// TIA Portal project "Szklarnia_AMN_V15.1" (V15.1)

(* hardware
DEVICE "S7-1200 station_1"  S7-1200 Station
   slot 0: "Rack_0"  Rack  V1.0
   slot 1: "PLC_1"  CPU 1212C AC/DC/Rly  6ES7 212-1BD30-0XB0  V2.2
   slot 101: "CM 1241 (RS232)_1"  6ES7 241-1AH30-0XB0  V1.0
DEVICE "HMI_1"  KTP600 Basic color PN
   slot 0: "HMI"  HMI  6AV6 647-0AD11-3AX0  12.0.0.0
   slot 1: "HMI_RT_1"  KTP600 Basic color PN  6AV6 647-0AD11-3AX0  12.0.0.0
   slot 5: "HMI_1.IE_CP_1"  PROFINET Interface
      slot 1: "PROFINET Interface_1"  PROFINET Interface
         slot 1: "Port_1"  Port
*)

// ===== PLC "PLC_1"  CPU 1212C AC/DC/Rly =====

VAR_GLOBAL   // PLC tag table "Default tag table"
   "System_Byte" AT %MB1 : Byte;
   "FirstScan" AT %M1.0 : Bool;
   "DiagStatusUpdate" AT %M1.1 : Bool;
   "AlwaysTRUE" AT %M1.2 : Bool;
   "AlwaysFALSE" AT %M1.3 : Bool;
   "Clock_Byte" AT %MB0 : Byte;
   "Clock_10Hz" AT %M0.0 : Bool;
   "Clock_5Hz" AT %M0.1 : Bool;
   "Clock_2.5Hz" AT %M0.2 : Bool;
   "Clock_2Hz" AT %M0.3 : Bool;
   "Clock_1.25Hz" AT %M0.4 : Bool;
   "Clock_1Hz" AT %M0.5 : Bool;
   "Clock_0.625Hz" AT %M0.6 : Bool;
   "Clock_0.5Hz" AT %M0.7 : Bool;
   "Sensor_nasłonecznienia" AT %IW64 : Word;
   "Tag_2" AT %I0.0 : Bool;
   "Rolety" AT %Q0.0 : Bool;
   "Czujnik" AT %IW66 : Int;
   "Okna" AT %Q0.1 : Bool;
   "Pompa_zbiornik" AT %Q0.2 : Bool;
   "Pompa_sieć" AT %Q0.3 : Bool;
   "Nawadnianie_strefa_1" AT %Q0.4 : Bool;
   "Nawadnianie_strefa_2" AT %Q0.5 : Bool;
   "Nawadnianie_strefa_3" AT %Q0.6 : Bool;
   "Nawadnianie_strefa_4" AT %Q0.7 : Bool;
END_VAR

DATA_BLOCK "Naslonecznienie_DB"   // DB1
{ S7_Optimized_Access := 'TRUE' }
AUTHOR : AMN
VERSION : 0.1
// stored: InstanceOfName Naslonecznienie
"Naslonecznienie"
BEGIN
END_DATA_BLOCK

DATA_BLOCK "Dane_programu"   // DB2
TITLE = Dane - zmienne
{ S7_Optimized_Access := 'TRUE' }
AUTHOR : AMN
VERSION : 0.1
// Zmienne dostępne dla całego programu.
   VAR
      blindShut : Bool := false;   // Stan rolet: 1 - zasłonięte, 0 - odsłonięte.
      Light_Lux_temp : Real;   // Wartość pomocnicza do działania programu - nasłonecznienie.
      lightLux_ : Real := 0.0;   // Nasłonecznienie.
      Temp_ : Real := 0.0;   // Temperatura.
      CO2_ : Real := 0.0;   // Poziom CO2.
      setCO2 : Real := 5.0;   // Docelowa wartość CO2.
      setCO2_ : Real := 50.0;   // Docelowa wartość CO2 z HMI.
      setTemp : Real := 5.0;   // Docelowa wartość temperatury.
      setTemp_ : Real := 50.0;   // Docelowa wartość temperatury z HMI.
      StopBtn : Bool := false;   // Wyłącznik awaryjny: 1 - aktywny (blokada wszytskiego), 0 - nieaktywny.
      WaterLevel : Real := 5.0;   // Minimalny poziom wody w zbiorniku.
      StopPodlewanie : Bool := false;   // Blokada podlewania stref: 1 - Blokada podlewania, 0 - Możliwe podlewanie.
      Strefa1 : Bool := false;   // Blokada podlewania strefy 1: 1 - Blokada podlewania, 0 - możliwe podlewanie.
      Strefa2 : Bool := false;   // Blokada podlewania strefy 2: 1 - Blokada podlewania, 0 - możliwe podlewanie.
      Strefa3 : Bool := false;   // Blokada podlewania strefy 3: 1 - Blokada podlewania, 0 - możliwe podlewanie.
      Strefa4 : Bool := false;   // Blokada podlewania strefy 4: 1 - Blokada podlewania, 0 - możliwe podlewanie.
      Strefa5 : Bool := false;   // Blokada podlewania strefy 5: 1 - Blokada podlewania, 0 - możliwe podlewanie.
      setHum_Strefa2 : Real := 5.0;   // Docelowa wartość wilgotności - Strefa 2.
      setHum_Strefa1 : Real := 5.0;   // Docelowa wartość wilgotności - Strefa 1.
      setHum_Strefa5 : Real := 5.0;   // Docelowa wartość wilgotności - Strefa 5.
      setHum_Strefa4 : Real := 5.0;   // Docelowa wartość wilgotności - Strefa 4.
      setHum_Strefa3 : Real := 5.0;   // Docelowa wartość wilgotności - Strefa 3.
      setHum_Strefa1_ : Real := 50.0;   // Docelowa wartość wilgotności z HMI - Strefa 1.
      setHum_Strefa2_ : Real := 50.0;   // Docelowa wartość wilgotności z HMI - Strefa 2.
      setHum_Strefa3_ : Real := 50.0;   // Docelowa wartość wilgotności z HMI - Strefa 3.
      setHum_Strefa4_ : Real := 50.0;   // Docelowa wartość wilgotności z HMI - Strefa 4.
      setHum_Strefa5_ : Real := 50.0;   // Docelowa wartość wilgotności z HMI - Strefa 5.
      Strefa1_podlewanie : Bool := false;   // Aktywne podlewanie strefy 1: 1 - podlewanie, 0 - nie podlewa.
      Strefa2_podlewanie : Bool := false;   // Aktywne podlewanie strefy 2: 1 - podlewanie, 0 - nie podlewa.
      Strefa3_podlewanie : Bool := false;   // Aktywne podlewanie strefy 3: 1 - podlewanie, 0 - nie podlewa.
      Strefa4_podlewanie : Bool := false;   // Aktywne podlewanie strefy 4: 1 - podlewanie, 0 - nie podlewa.
      Strefa5_podlewanie : Bool := false;   // Aktywne podlewanie strefy 5: 1 - podlewanie, 0 - nie podlewa.
      WinOpen : Bool := false;   // Stan okien: 1 - otwarte, 0 - zamknięte.
      setLux : Real := 5.0;   // Docelowa wartość oświetlenia.
      setLux_ : Real := 50.0;   // Docelowa wartość oświetlenia z HMI.
      Hum_Strefa5 : Real := 0.0;   // Wilgotność strefy 5.
      Hum_Strefa4 : Real := 0.0;   // Wilgotność strefy 4.
      Hum_Strefa3 : Real := 0.0;   // Wilgotność strefy 3.
      Hum_Strefa2 : Real := 0.0;   // Wilgotność strefy 2.
      Hum_Strefa1 : Real := 0.0;   // Wilgotność strefy 1.
      Lux_Start : Bool := true;   // Pomiar początkowy nasłonecznienia.
      Nasłonecznienie : Array[0..6] of Real;   // Akwizycja pomiarów do wizualizacji - nałonecznienie.
      CO2 : Array[0..6] of Real;   // Akwizycja pomiarów do wizualizacji - CO2.
      Temperatura : Array[0..6] of Real;   // Akwizycja pomiarów do wizualizacji - Temperatura.
      Hum_1 : Array[0..6] of Real;   // Akwizycja pomiarów do wizualizacji - wilgotność strefy 1.
      Hum_2 : Array[0..6] of Real;   // Akwizycja pomiarów do wizualizacji - wilgotność strefy 2.
      Hum_3 : Array[0..6] of Real;   // Akwizycja pomiarów do wizualizacji - wilgotność strefy 3.
      Hum_4 : Array[0..6] of Real;   // Akwizycja pomiarów do wizualizacji - wilgotność strefy 4.
      Hum_5 : Array[0..6] of Real;   // Akwizycja pomiarów do wizualizacji - wilgotność strefy 5.
   END_VAR
BEGIN
   Nasłonecznienie[0] := 30.0;
   Nasłonecznienie[1] := 35.0;
   Nasłonecznienie[2] := 70.0;
   Nasłonecznienie[3] := 60.0;
   Nasłonecznienie[4] := 75.0;
   Nasłonecznienie[5] := 25.0;
   Nasłonecznienie[6] := 10.0;
   CO2[0] := 10.0;
   CO2[1] := 11.0;
   CO2[2] := 15.0;
   CO2[3] := 8.0;
   CO2[4] := 7.0;
   CO2[5] := 10.0;
   CO2[6] := 11.0;
   Temperatura[0] := 15.0;
   Temperatura[1] := 16.0;
   Temperatura[2] := 20.0;
   Temperatura[3] := 19.0;
   Temperatura[4] := 21.0;
   Temperatura[5] := 22.2;
   Temperatura[6] := 23.4;
   Hum_1[0] := 10.0;
   Hum_1[1] := 20.0;
   Hum_1[2] := 30.0;
   Hum_1[3] := 40.0;
   Hum_1[4] := 50.0;
   Hum_1[5] := 50.0;
   Hum_1[6] := 60.0;
   Hum_2[0] := 90.0;
   Hum_2[1] := 80.0;
   Hum_2[2] := 44.4;
   Hum_2[3] := 34.3;
   Hum_2[4] := 77.7;
   Hum_2[5] := 78.8;
   Hum_2[6] := 80.0;
   Hum_3[0] := 33.3;
   Hum_3[1] := 56.6;
   Hum_3[2] := 76.7;
   Hum_3[3] := 87.8;
   Hum_3[4] := 98.9;
   Hum_3[5] := 12.1;
   Hum_3[6] := 45.4;
   Hum_4[0] := 66.6;
   Hum_4[1] := 77.7;
   Hum_4[2] := 65.6;
   Hum_4[3] := 55.5;
   Hum_4[4] := 55.5;
   Hum_4[5] := 55.5;
   Hum_4[6] := 66.4;
   Hum_5[0] := 23.4;
   Hum_5[1] := 34.5;
   Hum_5[2] := 53.5;
   Hum_5[3] := 98.7;
   Hum_5[4] := 54.3;
   Hum_5[5] := 56.9;
   Hum_5[6] := 22.2;
END_DATA_BLOCK

DATA_BLOCK "CO2_DB"   // DB8
{ S7_Optimized_Access := 'TRUE' }
AUTHOR : AMN
VERSION : 0.1
// stored: InstanceOfName CO2
"CO2"
BEGIN
END_DATA_BLOCK

DATA_BLOCK "Naslonecznienie_DB_1"   // DB9
{ S7_Optimized_Access := 'TRUE' }
AUTHOR : AMN
VERSION : 0.1
// stored: InstanceOfName Naslonecznienie
"Naslonecznienie"
BEGIN
END_DATA_BLOCK

DATA_BLOCK "CO2_DB_1"   // DB10
{ S7_Optimized_Access := 'TRUE' }
AUTHOR : AMN
VERSION : 0.1
// stored: InstanceOfName CO2
"CO2"
BEGIN
END_DATA_BLOCK

DATA_BLOCK "Temperature_DB"   // DB11
{ S7_Optimized_Access := 'TRUE' }
AUTHOR : AMN
VERSION : 0.1
// stored: InstanceOfName Temperature
"Temperature"
BEGIN
END_DATA_BLOCK

DATA_BLOCK "Nawadniane_DB"   // DB12
{ S7_Optimized_Access := 'TRUE' }
AUTHOR : AMN
VERSION : 0.1
// stored: InstanceOfName Nawadniane
"Nawadniane"
BEGIN
END_DATA_BLOCK

DATA_BLOCK "Nawadniane_DB_1"   // DB13
{ S7_Optimized_Access := 'TRUE' }
AUTHOR : AMN
VERSION : 0.1
// stored: InstanceOfName Nawadniane
"Nawadniane"
BEGIN
END_DATA_BLOCK

DATA_BLOCK "Nawadniane_DB_2"   // DB14
{ S7_Optimized_Access := 'TRUE' }
AUTHOR : AMN
VERSION : 0.1
// stored: InstanceOfName Nawadniane
"Nawadniane"
BEGIN
END_DATA_BLOCK

DATA_BLOCK "Nawadniane_DB_3"   // DB15
{ S7_Optimized_Access := 'TRUE' }
AUTHOR : AMN
VERSION : 0.1
// stored: InstanceOfName Nawadniane
"Nawadniane"
BEGIN
END_DATA_BLOCK

DATA_BLOCK "Nawadniane_DB_4"   // DB16
{ S7_Optimized_Access := 'TRUE' }
AUTHOR : AMN
VERSION : 0.1
// stored: InstanceOfName Nawadniane
"Nawadniane"
BEGIN
END_DATA_BLOCK

// folder: System blocks/Program resources

DATA_BLOCK "IEC_Timer_0_DB"   // DB3
{ S7_Optimized_Access := 'TRUE' }
AUTHOR : Simatic
FAMILY : IEC
NAME : IEC_TMR
VERSION : 1.0
// stored: InstanceOfName IEC_TIMER
"IEC_TIMER"
BEGIN
END_DATA_BLOCK

DATA_BLOCK "IEC_Timer_0_DB_1"   // DB4
{ S7_Optimized_Access := 'TRUE' }
AUTHOR : Simatic
FAMILY : IEC
NAME : IEC_TMR
VERSION : 1.0
// stored: InstanceOfName IEC_TIMER
"IEC_TIMER"
BEGIN
END_DATA_BLOCK

DATA_BLOCK "IEC_Timer_0_DB_2"   // DB5
{ S7_Optimized_Access := 'TRUE' }
AUTHOR : Simatic
FAMILY : IEC
NAME : IEC_TMR
VERSION : 1.0
// stored: InstanceOfName IEC_TIMER
"IEC_TIMER"
BEGIN
END_DATA_BLOCK

DATA_BLOCK "IEC_Timer_0_DB_3"   // DB6
{ S7_Optimized_Access := 'TRUE' }
AUTHOR : Simatic
FAMILY : IEC
NAME : IEC_TMR
VERSION : 1.0
// stored: InstanceOfName IEC_TIMER
"IEC_TIMER"
BEGIN
END_DATA_BLOCK

DATA_BLOCK "IEC_Timer_0_DB_4"   // DB7
{ S7_Optimized_Access := 'TRUE' }
AUTHOR : Simatic
FAMILY : IEC
NAME : IEC_TMR
VERSION : 1.0
// stored: InstanceOfName IEC_TIMER
"IEC_TIMER"
BEGIN
END_DATA_BLOCK

DATA_BLOCK "IEC_Timer_0_DB_5"   // DB17
{ S7_Optimized_Access := 'TRUE' }
AUTHOR : Simatic
FAMILY : IEC
NAME : IEC_TMR
VERSION : 1.0
// stored: InstanceOfName IEC_TIMER
"IEC_TIMER"
BEGIN
END_DATA_BLOCK

// folder: (top level)

FUNCTION_BLOCK "Naslonecznienie"   // FB1, LAD
TITLE = Naslonecznienie - rolety
{ S7_Optimized_Access := 'TRUE' }
AUTHOR : AMN
VERSION : 0.1
// Blok sterowania nasłonecznieniem - rolety
   VAR_INPUT
      lightLux_sensor : Int;
   END_VAR
   VAR_OUTPUT
      Rolety : Bool;   // True - zasłonięte, False - odsłonięte
   END_VAR
   VAR_TEMP
      lightLux_norm : Real;
      Galaz_TAK : Bool;
      lightLux : Real;
   END_VAR
   VAR_TEMP   // added for the SCL form of the ladder/FBD networks
      _w1 : Bool;
      _w2 : Bool;
   END_VAR
BEGIN

REGION Network 1: Odczytanie nasłoncznienia
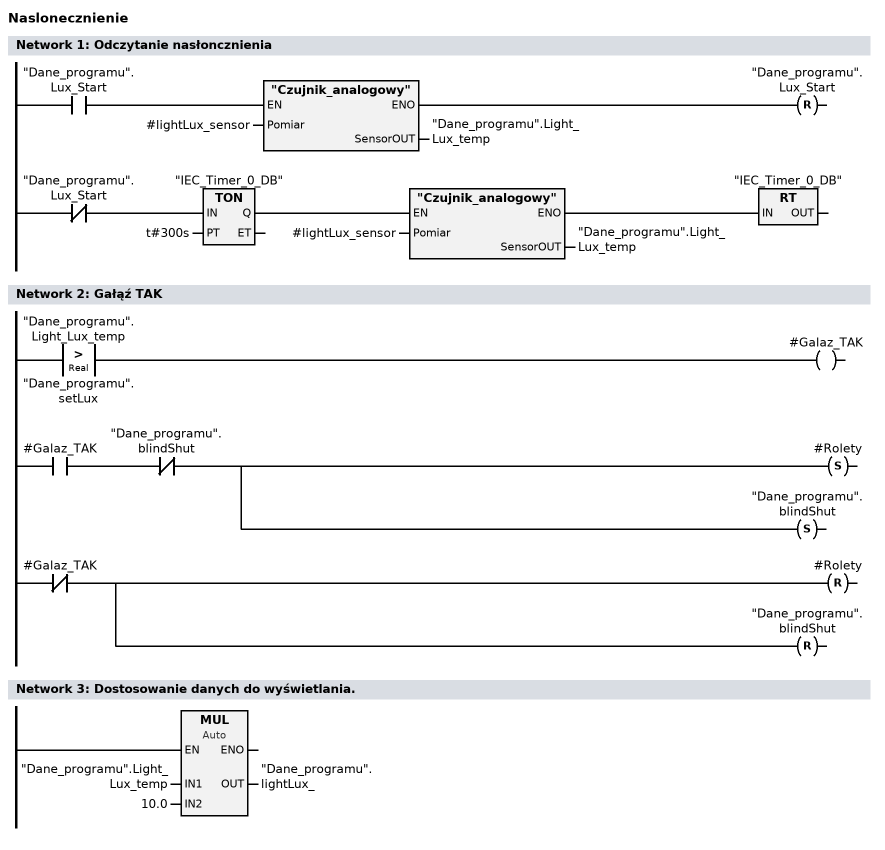
   "Czujnik_analogowy"(EN := "Dane_programu".Lux_Start,
                       Pomiar := #lightLux_sensor,
                       SensorOUT => "Dane_programu".Light_Lux_temp,
                       ENO => #_w1);
   IF #_w1 THEN "Dane_programu".Lux_Start := FALSE; END_IF;
   "IEC_Timer_0_DB".TON(IN := NOT "Dane_programu".Lux_Start, PT := t#300s);
   "Czujnik_analogowy"(EN := "IEC_Timer_0_DB".Q,
                       Pomiar := #lightLux_sensor,
                       SensorOUT => "Dane_programu".Light_Lux_temp,
                       ENO => #_w2);
   IF #_w2 THEN RESET_TIMER("IEC_Timer_0_DB"); END_IF;
END_REGION

REGION Network 2: Gałąź TAK
   RUNG wire#powerrail
      { S7_Templates := "SrcType := Real" } GT_Contact(in1 := "Dane_programu".Light_Lux_temp, in2 := "Dane_programu".setLux)
      Coil( #Galaz_TAK )
   END_RUNG
   RUNG wire#powerrail
      Contact( #Galaz_TAK )
      I_Contact( "Dane_programu".blindShut )
      wire#w1
      S_Coil( #Rolety )
   END_RUNG
   RUNG wire#w1
      S_Coil( "Dane_programu".blindShut )
   END_RUNG
   RUNG wire#powerrail
      I_Contact( #Galaz_TAK )
      wire#w2
      R_Coil( #Rolety )
   END_RUNG
   RUNG wire#w2
      R_Coil( "Dane_programu".blindShut )
   END_RUNG
   // the same network as SCL:
   #Galaz_TAK := "Dane_programu".Light_Lux_temp > "Dane_programu".setLux;
   IF #Galaz_TAK AND NOT "Dane_programu".blindShut THEN
       #Rolety := TRUE;
       "Dane_programu".blindShut := TRUE;
   END_IF;
   IF NOT #Galaz_TAK THEN
       #Rolety := FALSE;
       "Dane_programu".blindShut := FALSE;
   END_IF;
END_REGION

REGION Network 3: Dostosowanie danych do wyświetlania.
   RUNG wire#powerrail
      { S7_GenerateENO := "TRUE" } Mul(in1 := "Dane_programu".Light_Lux_temp, in2 := 10.0, out => "Dane_programu".lightLux_)
   END_RUNG
   // the same network as SCL:
   "Dane_programu".lightLux_ := "Dane_programu".Light_Lux_temp * 10.0;
END_REGION
END_FUNCTION_BLOCK

FUNCTION_BLOCK "CO2"   // FB2, LAD
TITLE = Sterowanie CO2
{ S7_Optimized_Access := 'TRUE' }
AUTHOR : AMN
VERSION : 0.1
// Schemat sterowania poziomem CO2
   VAR_INPUT
      CO2Sensor : Int;
   END_VAR
   VAR_OUTPUT
      Windows : Bool;   // True - otwarte, False - zamknięte
   END_VAR
   VAR_TEMP
      CO2_mes : Real;   // Wartość poziomu CO2
      temp1 : Bool;
      WinFlag : Bool;
   END_VAR
   VAR_TEMP   // added for the SCL form of the ladder/FBD networks
      _w1 : Bool;
   END_VAR
BEGIN

REGION Network 1
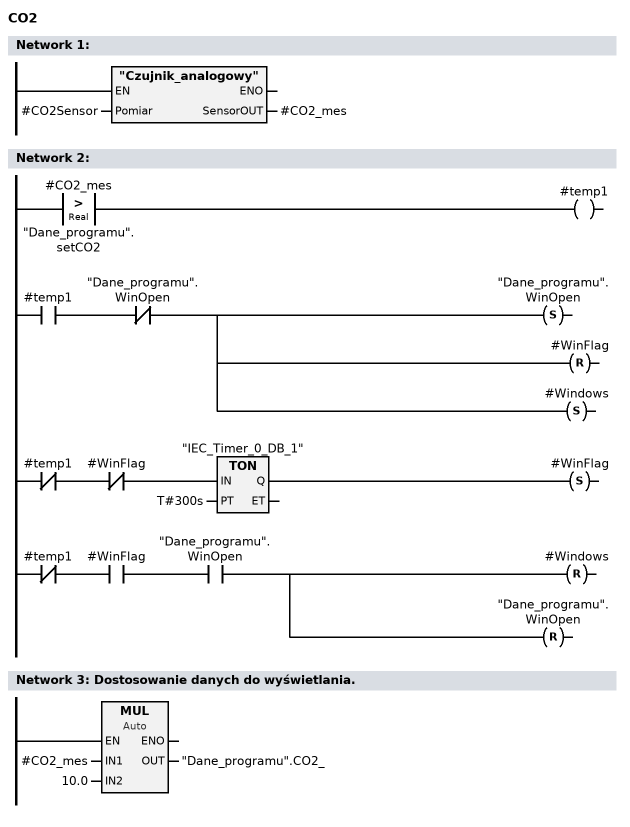
   RUNG wire#powerrail
      "Czujnik_analogowy"(Pomiar := #CO2Sensor, SensorOUT => #CO2_mes)
   END_RUNG
   // the same network as SCL:
   "Czujnik_analogowy"(Pomiar := #CO2Sensor, SensorOUT => #CO2_mes);
END_REGION

REGION Network 2
   #temp1 := #CO2_mes > "Dane_programu".setCO2;
   #_w1 := #temp1 AND NOT "Dane_programu".WinOpen;
   IF #_w1 THEN
       "Dane_programu".WinOpen := TRUE;
       #WinFlag := FALSE;
       #Windows := TRUE;
   END_IF;
   "IEC_Timer_0_DB_1".TON(IN := NOT #temp1 AND NOT #WinFlag, PT := T#300s);
   IF "IEC_Timer_0_DB_1".Q THEN #WinFlag := TRUE; END_IF;
   IF NOT #temp1 AND #WinFlag AND "Dane_programu".WinOpen THEN
       #Windows := FALSE;
       "Dane_programu".WinOpen := FALSE;
   END_IF;
END_REGION

REGION Network 3: Dostosowanie danych do wyświetlania.
   RUNG wire#powerrail
      { S7_GenerateENO := "TRUE" } Mul(in1 := #CO2_mes, in2 := 10.0, out => "Dane_programu".CO2_)
   END_RUNG
   // the same network as SCL:
   "Dane_programu".CO2_ := #CO2_mes * 10.0;
END_REGION
END_FUNCTION_BLOCK

FUNCTION_BLOCK "Temperature"   // FB3, LAD
TITLE = Sterowanie temperaturą
{ S7_Optimized_Access := 'TRUE' }
AUTHOR : AMN
VERSION : 0.1
// Schemat sterowania temperaturą
   VAR_INPUT
      TempSensor : Int;
   END_VAR
   VAR_OUTPUT
      Windows : Bool;   // True - otwarte, False - zamknięte
   END_VAR
   VAR_TEMP
      Temp_mes : Real;
      temp1 : Bool;
      WinFlag : Bool;
   END_VAR
   VAR_TEMP   // added for the SCL form of the ladder/FBD networks
      _w1 : Bool;
   END_VAR
BEGIN

REGION Network 1
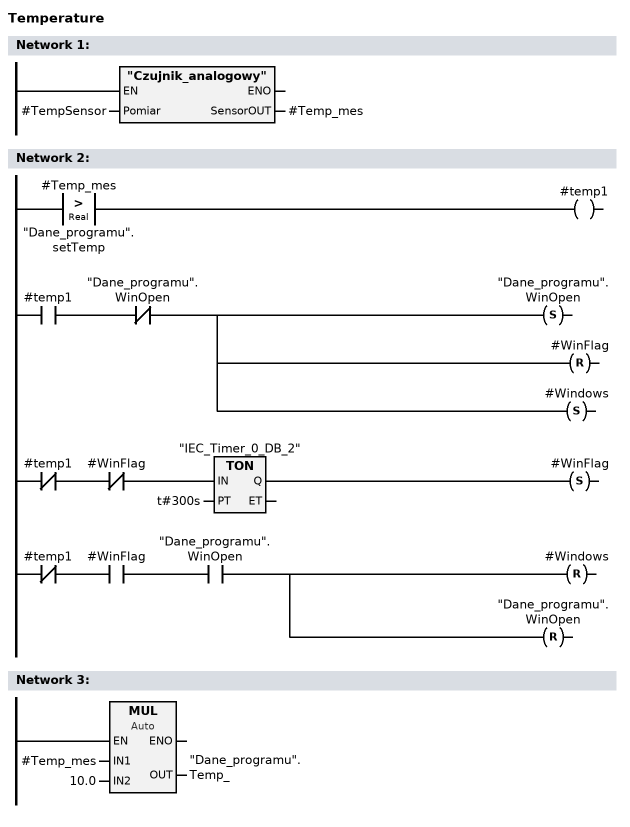
   RUNG wire#powerrail
      "Czujnik_analogowy"(Pomiar := #TempSensor, SensorOUT => #Temp_mes)
   END_RUNG
   // the same network as SCL:
   "Czujnik_analogowy"(Pomiar := #TempSensor, SensorOUT => #Temp_mes);
END_REGION

REGION Network 2
   #temp1 := #Temp_mes > "Dane_programu".setTemp;
   #_w1 := #temp1 AND NOT "Dane_programu".WinOpen;
   IF #_w1 THEN
       "Dane_programu".WinOpen := TRUE;
       #WinFlag := FALSE;
       #Windows := TRUE;
   END_IF;
   "IEC_Timer_0_DB_2".TON(IN := NOT #temp1 AND NOT #WinFlag, PT := t#300s);
   IF "IEC_Timer_0_DB_2".Q THEN #WinFlag := TRUE; END_IF;
   IF NOT #temp1 AND #WinFlag AND "Dane_programu".WinOpen THEN
       #Windows := FALSE;
       "Dane_programu".WinOpen := FALSE;
   END_IF;
END_REGION

REGION Network 3
   RUNG wire#powerrail
      { S7_GenerateENO := "TRUE" } Mul(in1 := #Temp_mes, in2 := 10.0, out => "Dane_programu".Temp_)
   END_RUNG
   // the same network as SCL:
   "Dane_programu".Temp_ := #Temp_mes * 10.0;
END_REGION
END_FUNCTION_BLOCK

FUNCTION_BLOCK "Nawadniane"   // FB4, LAD
TITLE = Sterowanie nawadnianiem
{ S7_Optimized_Access := 'TRUE' }
AUTHOR : AMN
VERSION : 0.1
// Schemat sterowania nawadnianiem
   VAR_INPUT
      HumSensor : Int;
      WaterSensor : Int;
      setHum : Real;
      Blokada_strefy : Bool;
   END_VAR
   VAR_OUTPUT
      Pompa_ze_zbiornika : Bool;
      Pompa_z_sieci : Bool;
      Nawadnianie : Bool;
   END_VAR
   VAR_IN_OUT
      To_HMI : Real;
   END_VAR
   VAR_TEMP
      Hum_mes : Real;
      Water_mes : Real;
      temp1 : Bool;
      temp2 : Bool;
      temp3 : Bool;
   END_VAR
BEGIN

REGION Network 1
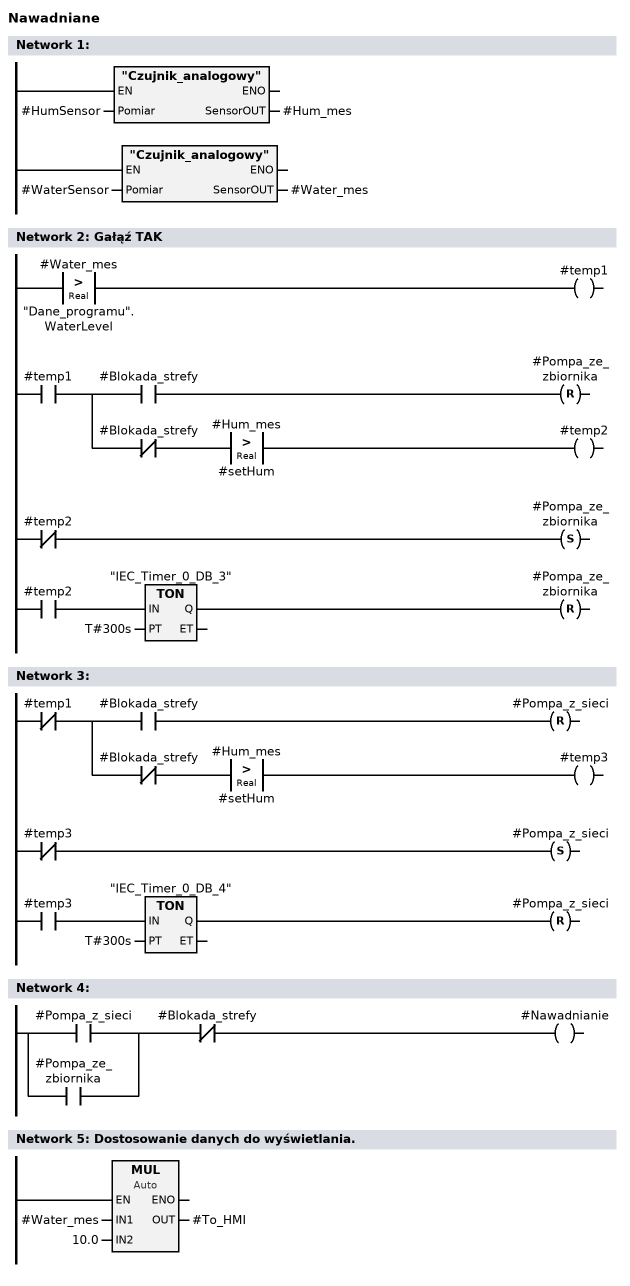
   RUNG wire#powerrail
      "Czujnik_analogowy"(Pomiar := #HumSensor, SensorOUT => #Hum_mes)
   END_RUNG
   RUNG wire#powerrail
      "Czujnik_analogowy"(Pomiar := #WaterSensor, SensorOUT => #Water_mes)
   END_RUNG
   // the same network as SCL:
   "Czujnik_analogowy"(Pomiar := #HumSensor, SensorOUT => #Hum_mes);
   "Czujnik_analogowy"(Pomiar := #WaterSensor, SensorOUT => #Water_mes);
END_REGION

REGION Network 2: Gałąź TAK
   #temp1 := #Water_mes > "Dane_programu".WaterLevel;
   IF #temp1 AND #Blokada_strefy THEN #Pompa_ze_zbiornika := FALSE; END_IF;
   #temp2 := #temp1 AND NOT #Blokada_strefy AND (#Hum_mes > #setHum);
   IF NOT #temp2 THEN #Pompa_ze_zbiornika := TRUE; END_IF;
   "IEC_Timer_0_DB_3".TON(IN := #temp2, PT := T#300s);
   IF "IEC_Timer_0_DB_3".Q THEN #Pompa_ze_zbiornika := FALSE; END_IF;
END_REGION

REGION Network 3
   IF NOT #temp1 AND #Blokada_strefy THEN #Pompa_z_sieci := FALSE; END_IF;
   #temp3 := NOT #temp1 AND NOT #Blokada_strefy AND (#Hum_mes > #setHum);
   IF NOT #temp3 THEN #Pompa_z_sieci := TRUE; END_IF;
   "IEC_Timer_0_DB_4".TON(IN := #temp3, PT := T#300s);
   IF "IEC_Timer_0_DB_4".Q THEN #Pompa_z_sieci := FALSE; END_IF;
END_REGION

REGION Network 4
   RUNG wire#powerrail
      Contact( #Pompa_z_sieci )
      wire#w1
      I_Contact( #Blokada_strefy )
      Coil( #Nawadnianie )
   END_RUNG
   RUNG wire#powerrail
      Contact( #Pompa_ze_zbiornika )
   END_RUNG wire#w1
   // the same network as SCL:
   #Nawadnianie := (#Pompa_z_sieci OR #Pompa_ze_zbiornika) AND NOT #Blokada_strefy;
END_REGION

REGION Network 5: Dostosowanie danych do wyświetlania.
   RUNG wire#powerrail
      { S7_GenerateENO := "TRUE" } Mul(in1 := #Water_mes, in2 := 10.0, out => #To_HMI)
   END_RUNG
   // the same network as SCL:
   #To_HMI := #Water_mes * 10.0;
END_REGION
END_FUNCTION_BLOCK

FUNCTION "Czujnik_analogowy" : Void   // FC1, LAD
TITLE = Pomiar z czujnika
{ S7_Optimized_Access := 'TRUE' }
AUTHOR : AMN
VERSION : 0.1
// Wyjście 0 - 10V
   VAR_INPUT
      Pomiar : Int;
   END_VAR
   VAR_OUTPUT
      SensorOUT : Real;
   END_VAR
   VAR_TEMP
      pomiar_norm : Real;
   END_VAR
BEGIN

REGION Network 1
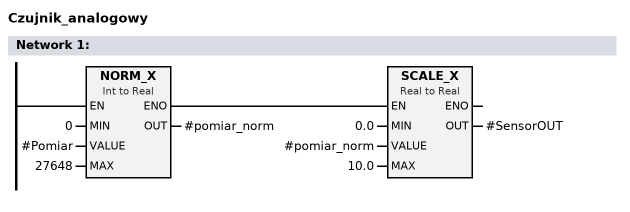
   RUNG wire#powerrail
      { S7_Templates := "[SrcType := Int, DestType := Real]"; S7_GenerateENO := "TRUE" } Normalize(min := 0, value := #Pomiar, max := 27648, out => #pomiar_norm)
      { S7_Templates := "[SrcType := Real, DestType := Real]"; S7_GenerateENO := "TRUE" } Scale(min := 0.0, value := #pomiar_norm, max := 10.0, out => #SensorOUT)
   END_RUNG
   // the same network as SCL:
   // ENO of a box is taken as its EN; it also drops when the box reports an error
   #pomiar_norm := NORM_X(MIN := 0, VALUE := #Pomiar, MAX := 27648);
   #SensorOUT := SCALE_X(MIN := 0.0, VALUE := #pomiar_norm, MAX := 10.0);
END_REGION
END_FUNCTION

FUNCTION "Program główny" : Void   // FC2, LAD
TITLE = Program główny
{ S7_Optimized_Access := 'TRUE' }
AUTHOR : AMN
VERSION : 0.1
// Schemat działania programu głównego.
   VAR_INPUT
      LightSensor : Int;
      CO2Sensor : Int;
      TempSensor : Int;
      WaterSensor : Int;
      HumSensor1 : Int;
      HumSensor2 : Int;
      HumSensor3 : Int;
      HumSensor4 : Int;
      HumSensor5 : Int;
   END_VAR
   VAR_OUTPUT
      Rolety : Bool;
      Okna : Bool;
      "Pompa ze zbiornika" : Bool;
      "Pompa z sieci" : Bool;
      Nawadnianie1 : Bool;
      Nawadnianie2 : Bool;
      Nawadnianie3 : Bool;
      Nawadnianie4 : Bool;
      Nawadnianie5 : Bool;
   END_VAR
   VAR_TEMP
      CO2_Win : Bool;
      Temp_Win : Bool;
   END_VAR
   VAR_TEMP   // added for the SCL form of the ladder/FBD networks
      _w1 : Bool;
   END_VAR
BEGIN

REGION Network 1: Nasłonecznienie, CO2, Temperaura
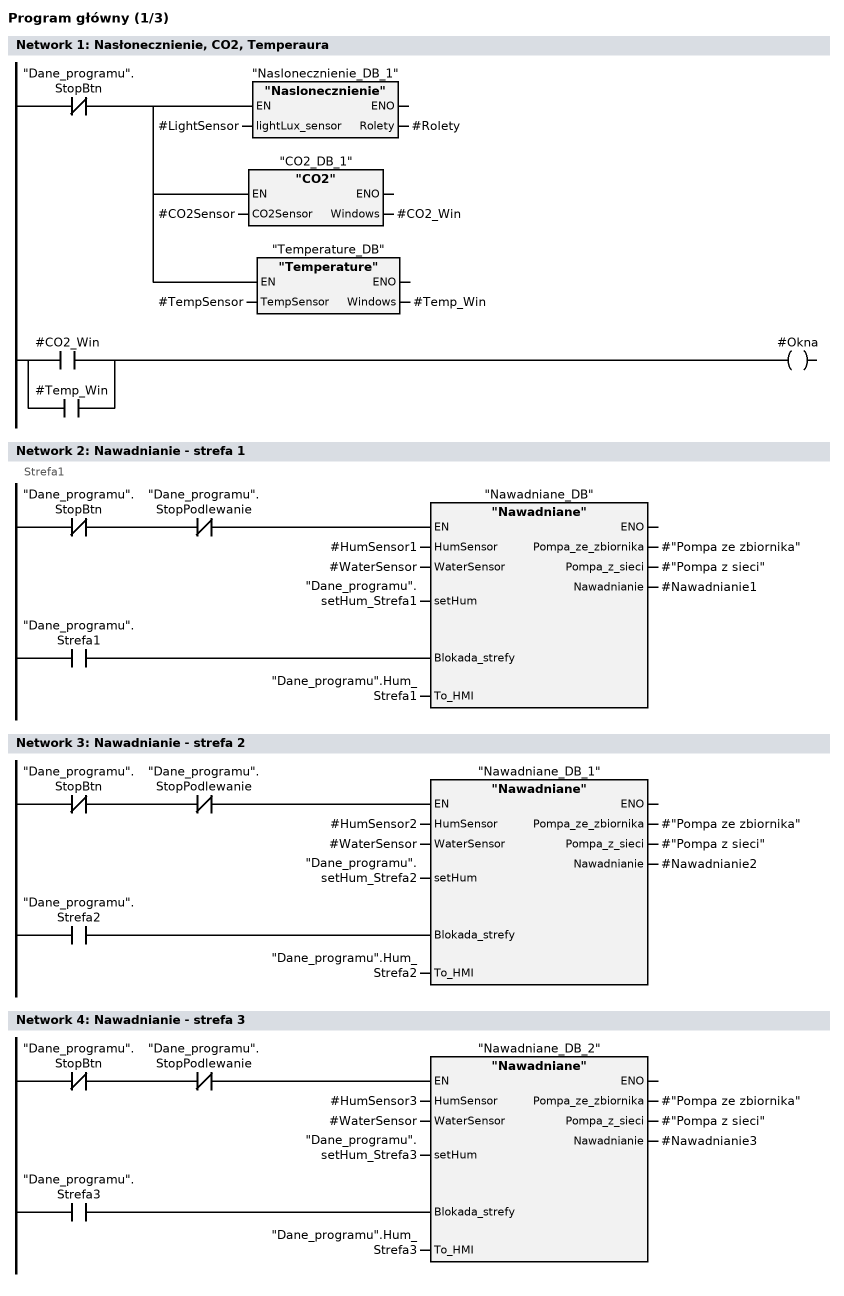
   RUNG wire#powerrail
      I_Contact( "Dane_programu".StopBtn )
      wire#w1
      "Naslonecznienie_DB_1"(lightLux_sensor := #LightSensor, Rolety => #Rolety)
   END_RUNG
   RUNG wire#w1
      "CO2_DB_1"(CO2Sensor := #CO2Sensor, Windows => #CO2_Win)
   END_RUNG
   RUNG wire#w1
      "Temperature_DB"(TempSensor := #TempSensor, Windows => #Temp_Win)
   END_RUNG
   RUNG wire#powerrail
      Contact( #CO2_Win )
      wire#w2
      Coil( #Okna )
   END_RUNG
   RUNG wire#powerrail
      Contact( #Temp_Win )
   END_RUNG wire#w2
   // the same network as SCL:
   #_w1 := NOT "Dane_programu".StopBtn;
   IF #_w1 THEN
       "Naslonecznienie_DB_1"(lightLux_sensor := #LightSensor, Rolety => #Rolety);   // "Naslonecznienie"
       "CO2_DB_1"(CO2Sensor := #CO2Sensor, Windows => #CO2_Win);   // "CO2"
       "Temperature_DB"(TempSensor := #TempSensor, Windows => #Temp_Win);   // "Temperature"
   END_IF;
   #Okna := #CO2_Win OR #Temp_Win;
END_REGION

REGION Network 2: Nawadnianie - strefa 1
   // Strefa1
   RUNG wire#powerrail
      I_Contact( "Dane_programu".StopBtn )
      I_Contact( "Dane_programu".StopPodlewanie )
      "Nawadniane_DB"(Blokada_strefy := wire#w1, HumSensor := #HumSensor1, WaterSensor := #WaterSensor, setHum := "Dane_programu".setHum_Strefa1, To_HMI := "Dane_programu".Hum_Strefa1, Pompa_ze_zbiornika => #"Pompa ze zbiornika", Pompa_z_sieci => #"Pompa z sieci", Nawadnianie => #Nawadnianie1)
   END_RUNG
   RUNG wire#powerrail
      Contact( "Dane_programu".Strefa1 )
   END_RUNG wire#w1
   // the same network as SCL:
   IF NOT "Dane_programu".StopBtn AND NOT "Dane_programu".StopPodlewanie THEN
       "Nawadniane_DB"(HumSensor := #HumSensor1,   // "Nawadniane"
                       WaterSensor := #WaterSensor,
                       setHum := "Dane_programu".setHum_Strefa1,
                       Blokada_strefy := "Dane_programu".Strefa1,
                       To_HMI := "Dane_programu".Hum_Strefa1,
                       Pompa_ze_zbiornika => #"Pompa ze zbiornika",
                       Pompa_z_sieci => #"Pompa z sieci",
                       Nawadnianie => #Nawadnianie1);
   END_IF;
END_REGION

REGION Network 3: Nawadnianie - strefa 2
   RUNG wire#powerrail
      I_Contact( "Dane_programu".StopBtn )
      I_Contact( "Dane_programu".StopPodlewanie )
      "Nawadniane_DB_1"(Blokada_strefy := wire#w1, HumSensor := #HumSensor2, WaterSensor := #WaterSensor, setHum := "Dane_programu".setHum_Strefa2, To_HMI := "Dane_programu".Hum_Strefa2, Pompa_ze_zbiornika => #"Pompa ze zbiornika", Pompa_z_sieci => #"Pompa z sieci", Nawadnianie => #Nawadnianie2)
   END_RUNG
   RUNG wire#powerrail
      Contact( "Dane_programu".Strefa2 )
   END_RUNG wire#w1
   // the same network as SCL:
   IF NOT "Dane_programu".StopBtn AND NOT "Dane_programu".StopPodlewanie THEN
       "Nawadniane_DB_1"(HumSensor := #HumSensor2,   // "Nawadniane"
                         WaterSensor := #WaterSensor,
                         setHum := "Dane_programu".setHum_Strefa2,
                         Blokada_strefy := "Dane_programu".Strefa2,
                         To_HMI := "Dane_programu".Hum_Strefa2,
                         Pompa_ze_zbiornika => #"Pompa ze zbiornika",
                         Pompa_z_sieci => #"Pompa z sieci",
                         Nawadnianie => #Nawadnianie2);
   END_IF;
END_REGION

REGION Network 4: Nawadnianie - strefa 3
   RUNG wire#powerrail
      I_Contact( "Dane_programu".StopBtn )
      I_Contact( "Dane_programu".StopPodlewanie )
      "Nawadniane_DB_2"(Blokada_strefy := wire#w1, HumSensor := #HumSensor3, WaterSensor := #WaterSensor, setHum := "Dane_programu".setHum_Strefa3, To_HMI := "Dane_programu".Hum_Strefa3, Pompa_ze_zbiornika => #"Pompa ze zbiornika", Pompa_z_sieci => #"Pompa z sieci", Nawadnianie => #Nawadnianie3)
   END_RUNG
   RUNG wire#powerrail
      Contact( "Dane_programu".Strefa3 )
   END_RUNG wire#w1
   // the same network as SCL:
   IF NOT "Dane_programu".StopBtn AND NOT "Dane_programu".StopPodlewanie THEN
       "Nawadniane_DB_2"(HumSensor := #HumSensor3,   // "Nawadniane"
                         WaterSensor := #WaterSensor,
                         setHum := "Dane_programu".setHum_Strefa3,
                         Blokada_strefy := "Dane_programu".Strefa3,
                         To_HMI := "Dane_programu".Hum_Strefa3,
                         Pompa_ze_zbiornika => #"Pompa ze zbiornika",
                         Pompa_z_sieci => #"Pompa z sieci",
                         Nawadnianie => #Nawadnianie3);
   END_IF;
END_REGION

REGION Network 5: Nawadnianie - strefa 4
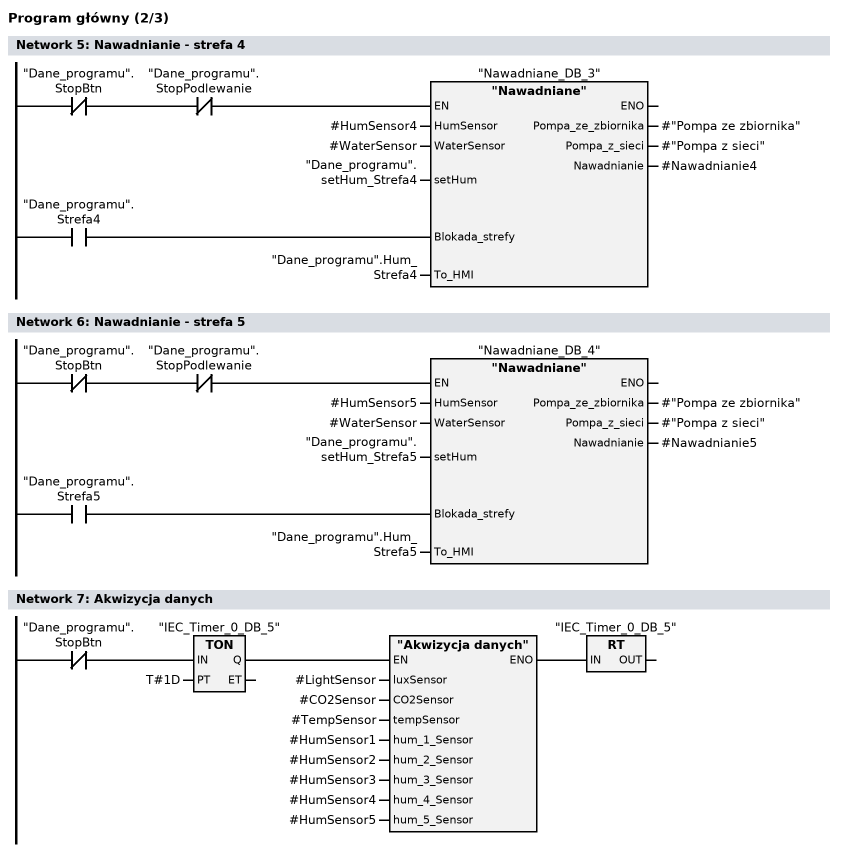
   RUNG wire#powerrail
      I_Contact( "Dane_programu".StopBtn )
      I_Contact( "Dane_programu".StopPodlewanie )
      "Nawadniane_DB_3"(Blokada_strefy := wire#w1, HumSensor := #HumSensor4, WaterSensor := #WaterSensor, setHum := "Dane_programu".setHum_Strefa4, To_HMI := "Dane_programu".Hum_Strefa4, Pompa_ze_zbiornika => #"Pompa ze zbiornika", Pompa_z_sieci => #"Pompa z sieci", Nawadnianie => #Nawadnianie4)
   END_RUNG
   RUNG wire#powerrail
      Contact( "Dane_programu".Strefa4 )
   END_RUNG wire#w1
   // the same network as SCL:
   IF NOT "Dane_programu".StopBtn AND NOT "Dane_programu".StopPodlewanie THEN
       "Nawadniane_DB_3"(HumSensor := #HumSensor4,   // "Nawadniane"
                         WaterSensor := #WaterSensor,
                         setHum := "Dane_programu".setHum_Strefa4,
                         Blokada_strefy := "Dane_programu".Strefa4,
                         To_HMI := "Dane_programu".Hum_Strefa4,
                         Pompa_ze_zbiornika => #"Pompa ze zbiornika",
                         Pompa_z_sieci => #"Pompa z sieci",
                         Nawadnianie => #Nawadnianie4);
   END_IF;
END_REGION

REGION Network 6: Nawadnianie - strefa 5
   RUNG wire#powerrail
      I_Contact( "Dane_programu".StopBtn )
      I_Contact( "Dane_programu".StopPodlewanie )
      "Nawadniane_DB_4"(Blokada_strefy := wire#w1, HumSensor := #HumSensor5, WaterSensor := #WaterSensor, setHum := "Dane_programu".setHum_Strefa5, To_HMI := "Dane_programu".Hum_Strefa5, Pompa_ze_zbiornika => #"Pompa ze zbiornika", Pompa_z_sieci => #"Pompa z sieci", Nawadnianie => #Nawadnianie5)
   END_RUNG
   RUNG wire#powerrail
      Contact( "Dane_programu".Strefa5 )
   END_RUNG wire#w1
   // the same network as SCL:
   IF NOT "Dane_programu".StopBtn AND NOT "Dane_programu".StopPodlewanie THEN
       "Nawadniane_DB_4"(HumSensor := #HumSensor5,   // "Nawadniane"
                         WaterSensor := #WaterSensor,
                         setHum := "Dane_programu".setHum_Strefa5,
                         Blokada_strefy := "Dane_programu".Strefa5,
                         To_HMI := "Dane_programu".Hum_Strefa5,
                         Pompa_ze_zbiornika => #"Pompa ze zbiornika",
                         Pompa_z_sieci => #"Pompa z sieci",
                         Nawadnianie => #Nawadnianie5);
   END_IF;
END_REGION

REGION Network 7: Akwizycja danych
   "IEC_Timer_0_DB_5".TON(IN := NOT "Dane_programu".StopBtn, PT := T#1D);
   "Akwizycja danych"(EN := "IEC_Timer_0_DB_5".Q,
                      luxSensor := #LightSensor,
                      CO2Sensor := #CO2Sensor,
                      tempSensor := #TempSensor,
                      hum_1_Sensor := #HumSensor1,
                      hum_2_Sensor := #HumSensor2,
                      hum_3_Sensor := #HumSensor3,
                      hum_4_Sensor := #HumSensor4,
                      hum_5_Sensor := #HumSensor5,
                      ENO => #_w1);
   IF #_w1 THEN RESET_TIMER("IEC_Timer_0_DB_5"); END_IF;
END_REGION

REGION Network 8: Dostosowanie z HMI do programu.
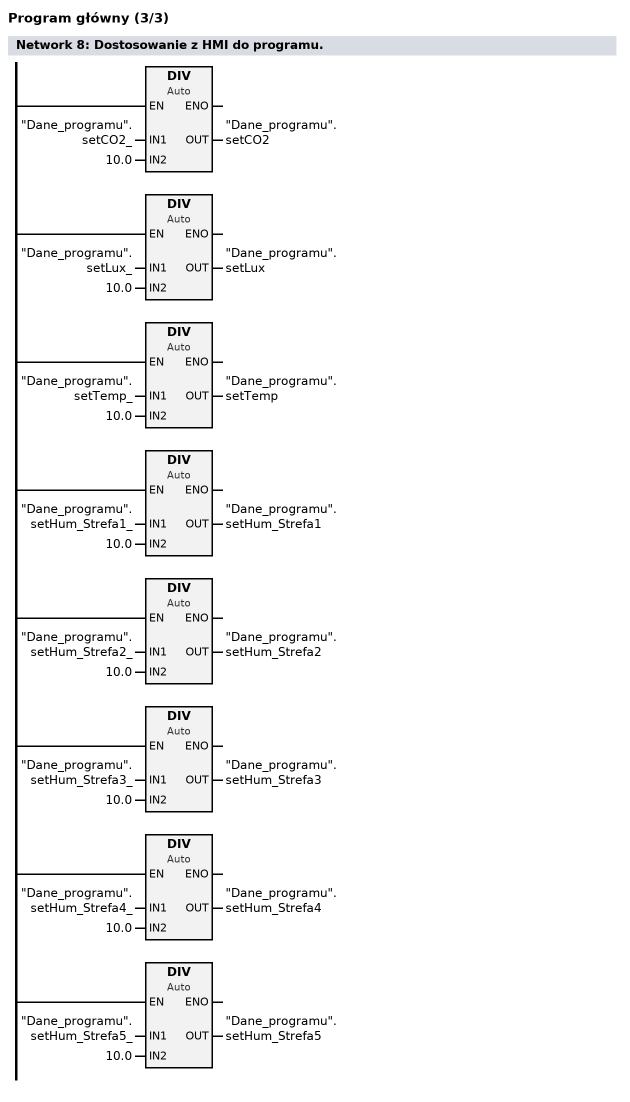
   RUNG wire#powerrail
      { S7_GenerateENO := "TRUE" } Div(in1 := "Dane_programu".setCO2_, in2 := 10.0, out => "Dane_programu".setCO2)
   END_RUNG
   RUNG wire#powerrail
      { S7_GenerateENO := "TRUE" } Div(in1 := "Dane_programu".setLux_, in2 := 10.0, out => "Dane_programu".setLux)
   END_RUNG
   RUNG wire#powerrail
      { S7_GenerateENO := "TRUE" } Div(in1 := "Dane_programu".setTemp_, in2 := 10.0, out => "Dane_programu".setTemp)
   END_RUNG
   RUNG wire#powerrail
      { S7_GenerateENO := "TRUE" } Div(in1 := "Dane_programu".setHum_Strefa1_, in2 := 10.0, out => "Dane_programu".setHum_Strefa1)
   END_RUNG
   RUNG wire#powerrail
      { S7_GenerateENO := "TRUE" } Div(in1 := "Dane_programu".setHum_Strefa2_, in2 := 10.0, out => "Dane_programu".setHum_Strefa2)
   END_RUNG
   RUNG wire#powerrail
      { S7_GenerateENO := "TRUE" } Div(in1 := "Dane_programu".setHum_Strefa3_, in2 := 10.0, out => "Dane_programu".setHum_Strefa3)
   END_RUNG
   RUNG wire#powerrail
      { S7_GenerateENO := "TRUE" } Div(in1 := "Dane_programu".setHum_Strefa4_, in2 := 10.0, out => "Dane_programu".setHum_Strefa4)
   END_RUNG
   RUNG wire#powerrail
      { S7_GenerateENO := "TRUE" } Div(in1 := "Dane_programu".setHum_Strefa5_, in2 := 10.0, out => "Dane_programu".setHum_Strefa5)
   END_RUNG
   // the same network as SCL:
   "Dane_programu".setCO2 := "Dane_programu".setCO2_ / 10.0;
   "Dane_programu".setLux := "Dane_programu".setLux_ / 10.0;
   "Dane_programu".setTemp := "Dane_programu".setTemp_ / 10.0;
   "Dane_programu".setHum_Strefa1 := "Dane_programu".setHum_Strefa1_ / 10.0;
   "Dane_programu".setHum_Strefa2 := "Dane_programu".setHum_Strefa2_ / 10.0;
   "Dane_programu".setHum_Strefa3 := "Dane_programu".setHum_Strefa3_ / 10.0;
   "Dane_programu".setHum_Strefa4 := "Dane_programu".setHum_Strefa4_ / 10.0;
   "Dane_programu".setHum_Strefa5 := "Dane_programu".setHum_Strefa5_ / 10.0;
END_REGION
END_FUNCTION

FUNCTION "Akwizycja danych" : Void   // FC3, LAD
TITLE = Program akwizycji danych do WebServera.
{ S7_Optimized_Access := 'TRUE' }
VERSION : 0.1
   VAR_INPUT
      luxSensor : Int;
      CO2Sensor : Int;
      tempSensor : Int;
      hum_1_Sensor : Int;
      hum_2_Sensor : Int;
      hum_3_Sensor : Int;
      hum_4_Sensor : Int;
      hum_5_Sensor : Int;
   END_VAR
   VAR_TEMP
      lux_mes : Real;
      co2_mes : Real;
      temp_mes : Real;
      hum_1_mes : Real;
      hum_2_mes : Real;
      hum_3_mes : Real;
      hum_4_mes : Real;
      hum_5_mes : Real;
   END_VAR
BEGIN

REGION Network 1: Nasłonecznienie
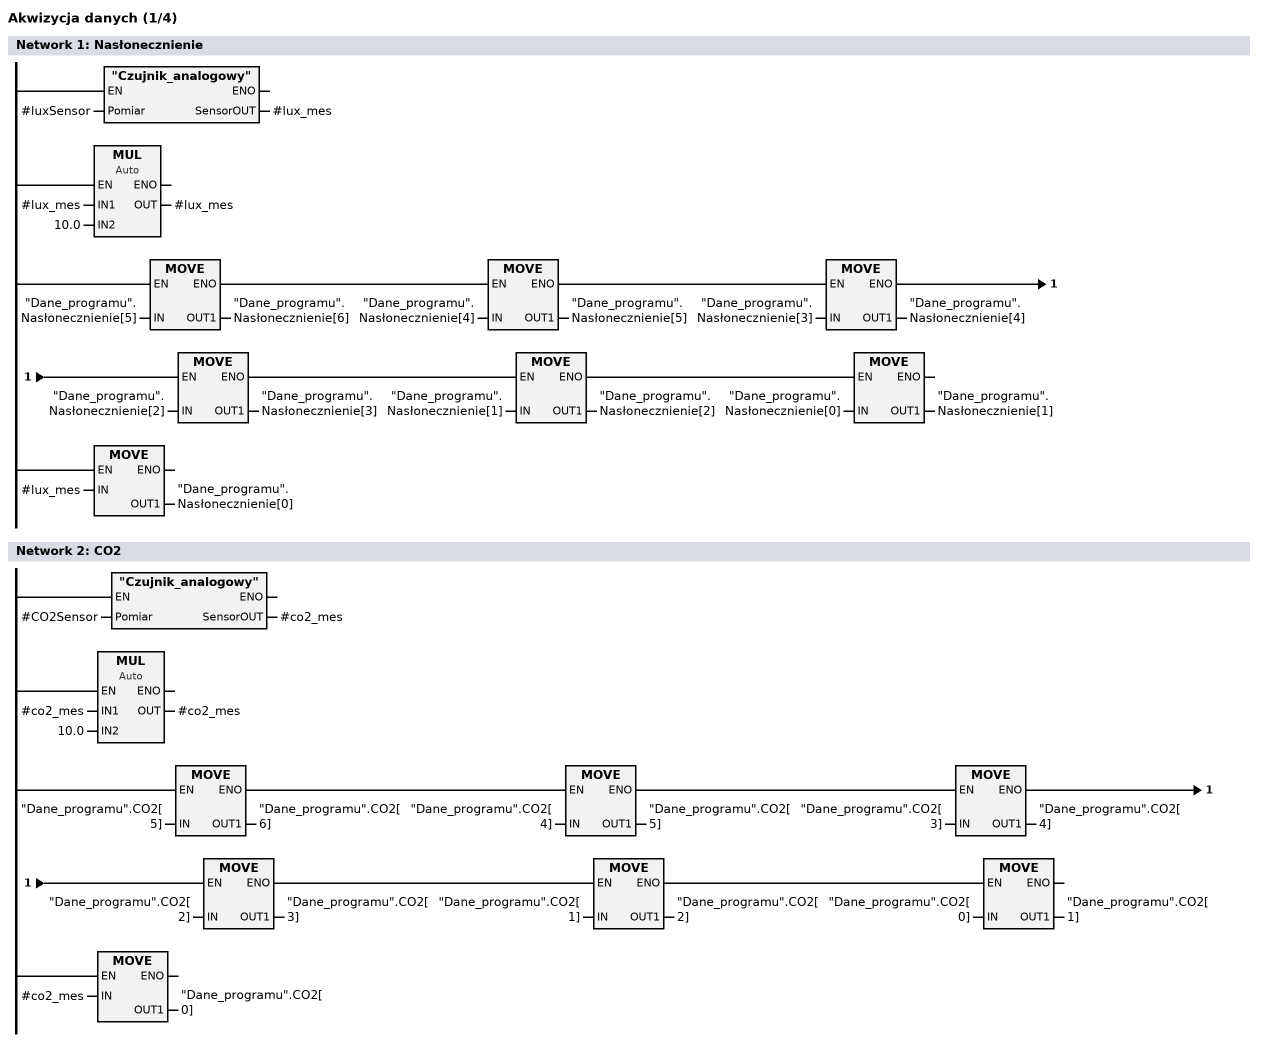
   RUNG wire#powerrail
      "Czujnik_analogowy"(Pomiar := #luxSensor, SensorOUT => #lux_mes)
   END_RUNG
   RUNG wire#powerrail
      { S7_GenerateENO := "TRUE" } Mul(in1 := #lux_mes, in2 := 10.0, out => #lux_mes)
   END_RUNG
   RUNG wire#powerrail
      { S7_GenerateENO := "TRUE" } Move(in := "Dane_programu".Nasłonecznienie[5], out1 => "Dane_programu".Nasłonecznienie[6])
      { S7_GenerateENO := "TRUE" } Move(in := "Dane_programu".Nasłonecznienie[4], out1 => "Dane_programu".Nasłonecznienie[5])
      { S7_GenerateENO := "TRUE" } Move(in := "Dane_programu".Nasłonecznienie[3], out1 => "Dane_programu".Nasłonecznienie[4])
      { S7_GenerateENO := "TRUE" } Move(in := "Dane_programu".Nasłonecznienie[2], out1 => "Dane_programu".Nasłonecznienie[3])
      { S7_GenerateENO := "TRUE" } Move(in := "Dane_programu".Nasłonecznienie[1], out1 => "Dane_programu".Nasłonecznienie[2])
      { S7_GenerateENO := "TRUE" } Move(in := "Dane_programu".Nasłonecznienie[0], out1 => "Dane_programu".Nasłonecznienie[1])
   END_RUNG
   RUNG wire#powerrail
      { S7_GenerateENO := "TRUE" } Move(in := #lux_mes, out1 => "Dane_programu".Nasłonecznienie[0])
   END_RUNG
   // the same network as SCL:
   // ENO of a box is taken as its EN; it also drops when the box reports an error
   "Czujnik_analogowy"(Pomiar := #luxSensor, SensorOUT => #lux_mes);
   #lux_mes := #lux_mes * 10.0;
   "Dane_programu".Nasłonecznienie[6] := "Dane_programu".Nasłonecznienie[5];
   "Dane_programu".Nasłonecznienie[5] := "Dane_programu".Nasłonecznienie[4];
   "Dane_programu".Nasłonecznienie[4] := "Dane_programu".Nasłonecznienie[3];
   "Dane_programu".Nasłonecznienie[3] := "Dane_programu".Nasłonecznienie[2];
   "Dane_programu".Nasłonecznienie[2] := "Dane_programu".Nasłonecznienie[1];
   "Dane_programu".Nasłonecznienie[1] := "Dane_programu".Nasłonecznienie[0];
   "Dane_programu".Nasłonecznienie[0] := #lux_mes;
END_REGION

REGION Network 2: CO2
   RUNG wire#powerrail
      "Czujnik_analogowy"(Pomiar := #CO2Sensor, SensorOUT => #co2_mes)
   END_RUNG
   RUNG wire#powerrail
      { S7_GenerateENO := "TRUE" } Mul(in1 := #co2_mes, in2 := 10.0, out => #co2_mes)
   END_RUNG
   RUNG wire#powerrail
      { S7_GenerateENO := "TRUE" } Move(in := "Dane_programu".CO2[5], out1 => "Dane_programu".CO2[6])
      { S7_GenerateENO := "TRUE" } Move(in := "Dane_programu".CO2[4], out1 => "Dane_programu".CO2[5])
      { S7_GenerateENO := "TRUE" } Move(in := "Dane_programu".CO2[3], out1 => "Dane_programu".CO2[4])
      { S7_GenerateENO := "TRUE" } Move(in := "Dane_programu".CO2[2], out1 => "Dane_programu".CO2[3])
      { S7_GenerateENO := "TRUE" } Move(in := "Dane_programu".CO2[1], out1 => "Dane_programu".CO2[2])
      { S7_GenerateENO := "TRUE" } Move(in := "Dane_programu".CO2[0], out1 => "Dane_programu".CO2[1])
   END_RUNG
   RUNG wire#powerrail
      { S7_GenerateENO := "TRUE" } Move(in := #co2_mes, out1 => "Dane_programu".CO2[0])
   END_RUNG
   // the same network as SCL:
   // ENO of a box is taken as its EN; it also drops when the box reports an error
   "Czujnik_analogowy"(Pomiar := #CO2Sensor, SensorOUT => #co2_mes);
   #co2_mes := #co2_mes * 10.0;
   "Dane_programu".CO2[6] := "Dane_programu".CO2[5];
   "Dane_programu".CO2[5] := "Dane_programu".CO2[4];
   "Dane_programu".CO2[4] := "Dane_programu".CO2[3];
   "Dane_programu".CO2[3] := "Dane_programu".CO2[2];
   "Dane_programu".CO2[2] := "Dane_programu".CO2[1];
   "Dane_programu".CO2[1] := "Dane_programu".CO2[0];
   "Dane_programu".CO2[0] := #co2_mes;
END_REGION

REGION Network 3: Temperature
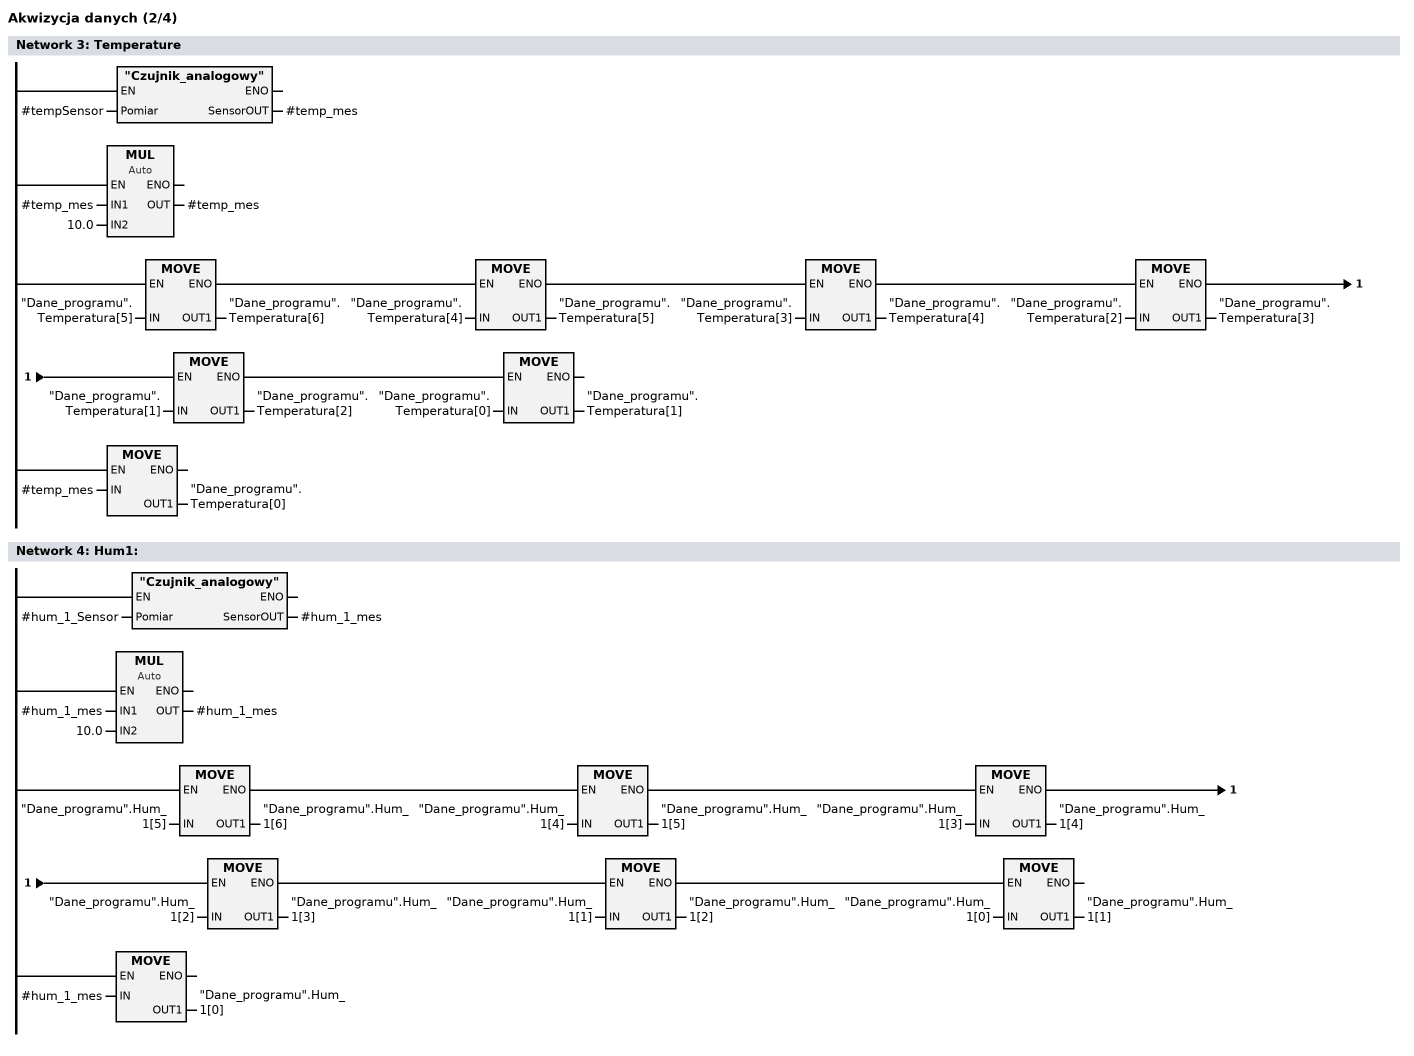
   RUNG wire#powerrail
      "Czujnik_analogowy"(Pomiar := #tempSensor, SensorOUT => #temp_mes)
   END_RUNG
   RUNG wire#powerrail
      { S7_GenerateENO := "TRUE" } Mul(in1 := #temp_mes, in2 := 10.0, out => #temp_mes)
   END_RUNG
   RUNG wire#powerrail
      { S7_GenerateENO := "TRUE" } Move(in := "Dane_programu".Temperatura[5], out1 => "Dane_programu".Temperatura[6])
      { S7_GenerateENO := "TRUE" } Move(in := "Dane_programu".Temperatura[4], out1 => "Dane_programu".Temperatura[5])
      { S7_GenerateENO := "TRUE" } Move(in := "Dane_programu".Temperatura[3], out1 => "Dane_programu".Temperatura[4])
      { S7_GenerateENO := "TRUE" } Move(in := "Dane_programu".Temperatura[2], out1 => "Dane_programu".Temperatura[3])
      { S7_GenerateENO := "TRUE" } Move(in := "Dane_programu".Temperatura[1], out1 => "Dane_programu".Temperatura[2])
      { S7_GenerateENO := "TRUE" } Move(in := "Dane_programu".Temperatura[0], out1 => "Dane_programu".Temperatura[1])
   END_RUNG
   RUNG wire#powerrail
      { S7_GenerateENO := "TRUE" } Move(in := #temp_mes, out1 => "Dane_programu".Temperatura[0])
   END_RUNG
   // the same network as SCL:
   // ENO of a box is taken as its EN; it also drops when the box reports an error
   "Czujnik_analogowy"(Pomiar := #tempSensor, SensorOUT => #temp_mes);
   #temp_mes := #temp_mes * 10.0;
   "Dane_programu".Temperatura[6] := "Dane_programu".Temperatura[5];
   "Dane_programu".Temperatura[5] := "Dane_programu".Temperatura[4];
   "Dane_programu".Temperatura[4] := "Dane_programu".Temperatura[3];
   "Dane_programu".Temperatura[3] := "Dane_programu".Temperatura[2];
   "Dane_programu".Temperatura[2] := "Dane_programu".Temperatura[1];
   "Dane_programu".Temperatura[1] := "Dane_programu".Temperatura[0];
   "Dane_programu".Temperatura[0] := #temp_mes;
END_REGION

REGION Network 4: Hum1:
   RUNG wire#powerrail
      "Czujnik_analogowy"(Pomiar := #hum_1_Sensor, SensorOUT => #hum_1_mes)
   END_RUNG
   RUNG wire#powerrail
      { S7_GenerateENO := "TRUE" } Mul(in1 := #hum_1_mes, in2 := 10.0, out => #hum_1_mes)
   END_RUNG
   RUNG wire#powerrail
      { S7_GenerateENO := "TRUE" } Move(in := "Dane_programu".Hum_1[5], out1 => "Dane_programu".Hum_1[6])
      { S7_GenerateENO := "TRUE" } Move(in := "Dane_programu".Hum_1[4], out1 => "Dane_programu".Hum_1[5])
      { S7_GenerateENO := "TRUE" } Move(in := "Dane_programu".Hum_1[3], out1 => "Dane_programu".Hum_1[4])
      { S7_GenerateENO := "TRUE" } Move(in := "Dane_programu".Hum_1[2], out1 => "Dane_programu".Hum_1[3])
      { S7_GenerateENO := "TRUE" } Move(in := "Dane_programu".Hum_1[1], out1 => "Dane_programu".Hum_1[2])
      { S7_GenerateENO := "TRUE" } Move(in := "Dane_programu".Hum_1[0], out1 => "Dane_programu".Hum_1[1])
   END_RUNG
   RUNG wire#powerrail
      { S7_GenerateENO := "TRUE" } Move(in := #hum_1_mes, out1 => "Dane_programu".Hum_1[0])
   END_RUNG
   // the same network as SCL:
   // ENO of a box is taken as its EN; it also drops when the box reports an error
   "Czujnik_analogowy"(Pomiar := #hum_1_Sensor, SensorOUT => #hum_1_mes);
   #hum_1_mes := #hum_1_mes * 10.0;
   "Dane_programu".Hum_1[6] := "Dane_programu".Hum_1[5];
   "Dane_programu".Hum_1[5] := "Dane_programu".Hum_1[4];
   "Dane_programu".Hum_1[4] := "Dane_programu".Hum_1[3];
   "Dane_programu".Hum_1[3] := "Dane_programu".Hum_1[2];
   "Dane_programu".Hum_1[2] := "Dane_programu".Hum_1[1];
   "Dane_programu".Hum_1[1] := "Dane_programu".Hum_1[0];
   "Dane_programu".Hum_1[0] := #hum_1_mes;
END_REGION

REGION Network 5: Hum2:
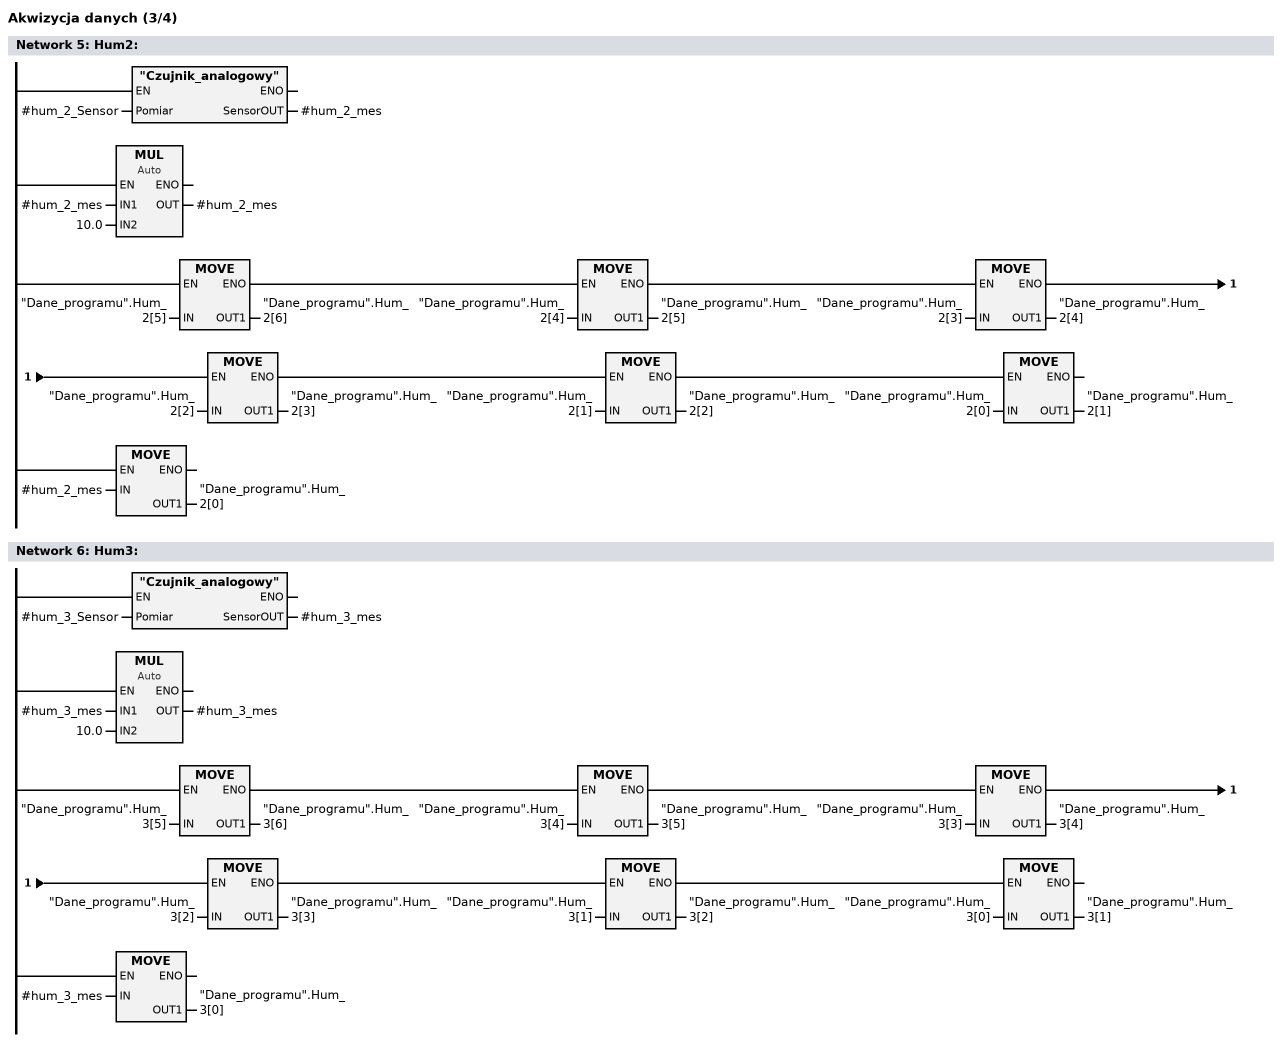
   RUNG wire#powerrail
      "Czujnik_analogowy"(Pomiar := #hum_2_Sensor, SensorOUT => #hum_2_mes)
   END_RUNG
   RUNG wire#powerrail
      { S7_GenerateENO := "TRUE" } Mul(in1 := #hum_2_mes, in2 := 10.0, out => #hum_2_mes)
   END_RUNG
   RUNG wire#powerrail
      { S7_GenerateENO := "TRUE" } Move(in := "Dane_programu".Hum_2[5], out1 => "Dane_programu".Hum_2[6])
      { S7_GenerateENO := "TRUE" } Move(in := "Dane_programu".Hum_2[4], out1 => "Dane_programu".Hum_2[5])
      { S7_GenerateENO := "TRUE" } Move(in := "Dane_programu".Hum_2[3], out1 => "Dane_programu".Hum_2[4])
      { S7_GenerateENO := "TRUE" } Move(in := "Dane_programu".Hum_2[2], out1 => "Dane_programu".Hum_2[3])
      { S7_GenerateENO := "TRUE" } Move(in := "Dane_programu".Hum_2[1], out1 => "Dane_programu".Hum_2[2])
      { S7_GenerateENO := "TRUE" } Move(in := "Dane_programu".Hum_2[0], out1 => "Dane_programu".Hum_2[1])
   END_RUNG
   RUNG wire#powerrail
      { S7_GenerateENO := "TRUE" } Move(in := #hum_2_mes, out1 => "Dane_programu".Hum_2[0])
   END_RUNG
   // the same network as SCL:
   // ENO of a box is taken as its EN; it also drops when the box reports an error
   "Czujnik_analogowy"(Pomiar := #hum_2_Sensor, SensorOUT => #hum_2_mes);
   #hum_2_mes := #hum_2_mes * 10.0;
   "Dane_programu".Hum_2[6] := "Dane_programu".Hum_2[5];
   "Dane_programu".Hum_2[5] := "Dane_programu".Hum_2[4];
   "Dane_programu".Hum_2[4] := "Dane_programu".Hum_2[3];
   "Dane_programu".Hum_2[3] := "Dane_programu".Hum_2[2];
   "Dane_programu".Hum_2[2] := "Dane_programu".Hum_2[1];
   "Dane_programu".Hum_2[1] := "Dane_programu".Hum_2[0];
   "Dane_programu".Hum_2[0] := #hum_2_mes;
END_REGION

REGION Network 6: Hum3:
   RUNG wire#powerrail
      "Czujnik_analogowy"(Pomiar := #hum_3_Sensor, SensorOUT => #hum_3_mes)
   END_RUNG
   RUNG wire#powerrail
      { S7_GenerateENO := "TRUE" } Mul(in1 := #hum_3_mes, in2 := 10.0, out => #hum_3_mes)
   END_RUNG
   RUNG wire#powerrail
      { S7_GenerateENO := "TRUE" } Move(in := "Dane_programu".Hum_3[5], out1 => "Dane_programu".Hum_3[6])
      { S7_GenerateENO := "TRUE" } Move(in := "Dane_programu".Hum_3[4], out1 => "Dane_programu".Hum_3[5])
      { S7_GenerateENO := "TRUE" } Move(in := "Dane_programu".Hum_3[3], out1 => "Dane_programu".Hum_3[4])
      { S7_GenerateENO := "TRUE" } Move(in := "Dane_programu".Hum_3[2], out1 => "Dane_programu".Hum_3[3])
      { S7_GenerateENO := "TRUE" } Move(in := "Dane_programu".Hum_3[1], out1 => "Dane_programu".Hum_3[2])
      { S7_GenerateENO := "TRUE" } Move(in := "Dane_programu".Hum_3[0], out1 => "Dane_programu".Hum_3[1])
   END_RUNG
   RUNG wire#powerrail
      { S7_GenerateENO := "TRUE" } Move(in := #hum_3_mes, out1 => "Dane_programu".Hum_3[0])
   END_RUNG
   // the same network as SCL:
   // ENO of a box is taken as its EN; it also drops when the box reports an error
   "Czujnik_analogowy"(Pomiar := #hum_3_Sensor, SensorOUT => #hum_3_mes);
   #hum_3_mes := #hum_3_mes * 10.0;
   "Dane_programu".Hum_3[6] := "Dane_programu".Hum_3[5];
   "Dane_programu".Hum_3[5] := "Dane_programu".Hum_3[4];
   "Dane_programu".Hum_3[4] := "Dane_programu".Hum_3[3];
   "Dane_programu".Hum_3[3] := "Dane_programu".Hum_3[2];
   "Dane_programu".Hum_3[2] := "Dane_programu".Hum_3[1];
   "Dane_programu".Hum_3[1] := "Dane_programu".Hum_3[0];
   "Dane_programu".Hum_3[0] := #hum_3_mes;
END_REGION

REGION Network 7: Hum4:
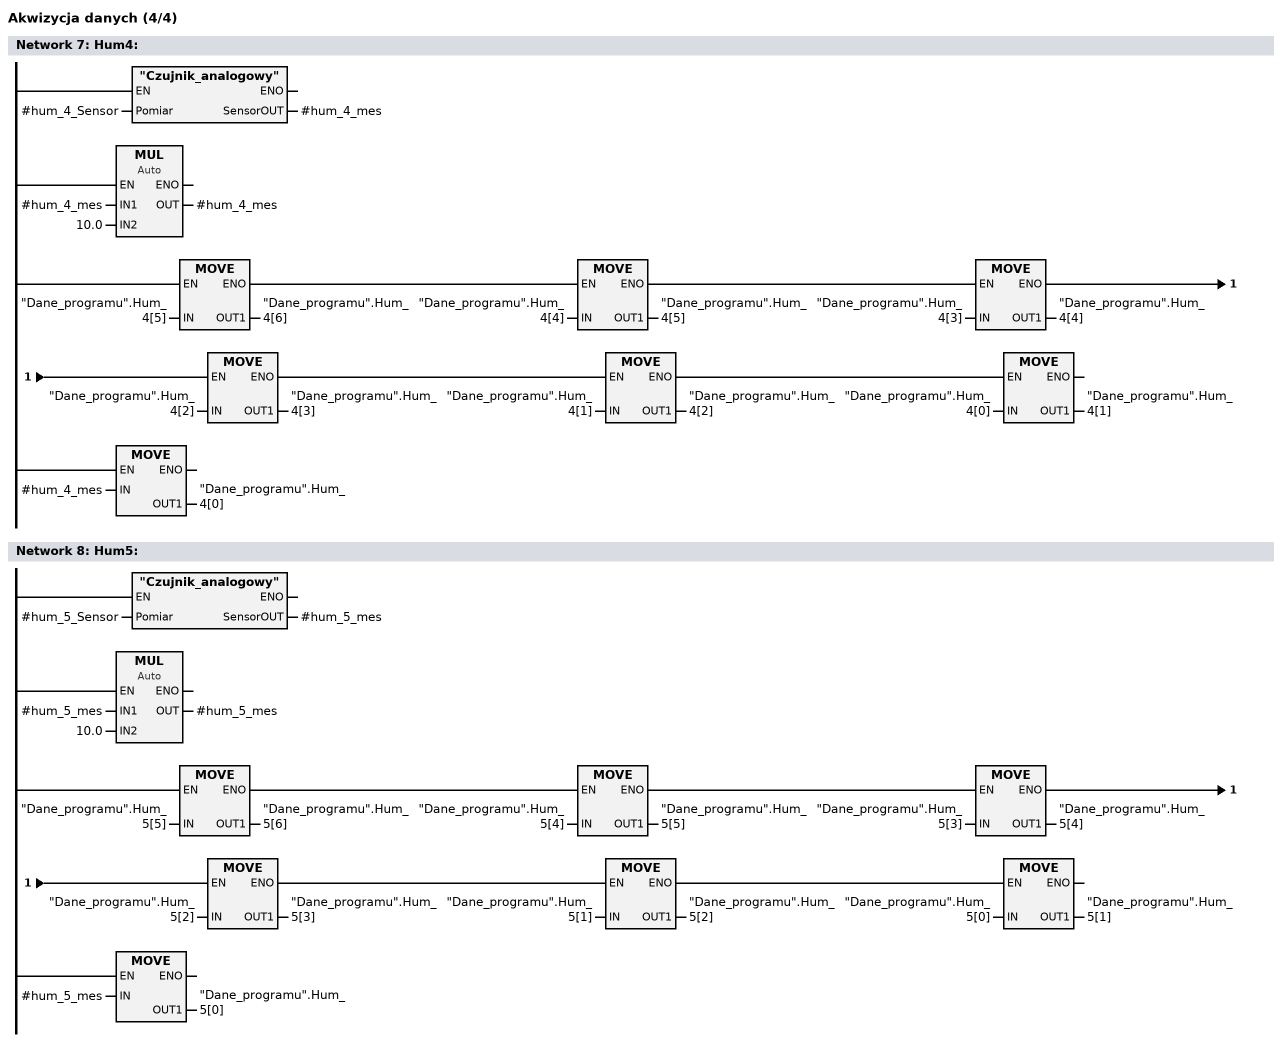
   RUNG wire#powerrail
      "Czujnik_analogowy"(Pomiar := #hum_4_Sensor, SensorOUT => #hum_4_mes)
   END_RUNG
   RUNG wire#powerrail
      { S7_GenerateENO := "TRUE" } Mul(in1 := #hum_4_mes, in2 := 10.0, out => #hum_4_mes)
   END_RUNG
   RUNG wire#powerrail
      { S7_GenerateENO := "TRUE" } Move(in := "Dane_programu".Hum_4[5], out1 => "Dane_programu".Hum_4[6])
      { S7_GenerateENO := "TRUE" } Move(in := "Dane_programu".Hum_4[4], out1 => "Dane_programu".Hum_4[5])
      { S7_GenerateENO := "TRUE" } Move(in := "Dane_programu".Hum_4[3], out1 => "Dane_programu".Hum_4[4])
      { S7_GenerateENO := "TRUE" } Move(in := "Dane_programu".Hum_4[2], out1 => "Dane_programu".Hum_4[3])
      { S7_GenerateENO := "TRUE" } Move(in := "Dane_programu".Hum_4[1], out1 => "Dane_programu".Hum_4[2])
      { S7_GenerateENO := "TRUE" } Move(in := "Dane_programu".Hum_4[0], out1 => "Dane_programu".Hum_4[1])
   END_RUNG
   RUNG wire#powerrail
      { S7_GenerateENO := "TRUE" } Move(in := #hum_4_mes, out1 => "Dane_programu".Hum_4[0])
   END_RUNG
   // the same network as SCL:
   // ENO of a box is taken as its EN; it also drops when the box reports an error
   "Czujnik_analogowy"(Pomiar := #hum_4_Sensor, SensorOUT => #hum_4_mes);
   #hum_4_mes := #hum_4_mes * 10.0;
   "Dane_programu".Hum_4[6] := "Dane_programu".Hum_4[5];
   "Dane_programu".Hum_4[5] := "Dane_programu".Hum_4[4];
   "Dane_programu".Hum_4[4] := "Dane_programu".Hum_4[3];
   "Dane_programu".Hum_4[3] := "Dane_programu".Hum_4[2];
   "Dane_programu".Hum_4[2] := "Dane_programu".Hum_4[1];
   "Dane_programu".Hum_4[1] := "Dane_programu".Hum_4[0];
   "Dane_programu".Hum_4[0] := #hum_4_mes;
END_REGION

REGION Network 8: Hum5:
   RUNG wire#powerrail
      "Czujnik_analogowy"(Pomiar := #hum_5_Sensor, SensorOUT => #hum_5_mes)
   END_RUNG
   RUNG wire#powerrail
      { S7_GenerateENO := "TRUE" } Mul(in1 := #hum_5_mes, in2 := 10.0, out => #hum_5_mes)
   END_RUNG
   RUNG wire#powerrail
      { S7_GenerateENO := "TRUE" } Move(in := "Dane_programu".Hum_5[5], out1 => "Dane_programu".Hum_5[6])
      { S7_GenerateENO := "TRUE" } Move(in := "Dane_programu".Hum_5[4], out1 => "Dane_programu".Hum_5[5])
      { S7_GenerateENO := "TRUE" } Move(in := "Dane_programu".Hum_5[3], out1 => "Dane_programu".Hum_5[4])
      { S7_GenerateENO := "TRUE" } Move(in := "Dane_programu".Hum_5[2], out1 => "Dane_programu".Hum_5[3])
      { S7_GenerateENO := "TRUE" } Move(in := "Dane_programu".Hum_5[1], out1 => "Dane_programu".Hum_5[2])
      { S7_GenerateENO := "TRUE" } Move(in := "Dane_programu".Hum_5[0], out1 => "Dane_programu".Hum_5[1])
   END_RUNG
   RUNG wire#powerrail
      { S7_GenerateENO := "TRUE" } Move(in := #hum_5_mes, out1 => "Dane_programu".Hum_5[0])
   END_RUNG
   // the same network as SCL:
   // ENO of a box is taken as its EN; it also drops when the box reports an error
   "Czujnik_analogowy"(Pomiar := #hum_5_Sensor, SensorOUT => #hum_5_mes);
   #hum_5_mes := #hum_5_mes * 10.0;
   "Dane_programu".Hum_5[6] := "Dane_programu".Hum_5[5];
   "Dane_programu".Hum_5[5] := "Dane_programu".Hum_5[4];
   "Dane_programu".Hum_5[4] := "Dane_programu".Hum_5[3];
   "Dane_programu".Hum_5[3] := "Dane_programu".Hum_5[2];
   "Dane_programu".Hum_5[2] := "Dane_programu".Hum_5[1];
   "Dane_programu".Hum_5[1] := "Dane_programu".Hum_5[0];
   "Dane_programu".Hum_5[0] := #hum_5_mes;
END_REGION
END_FUNCTION

ORGANIZATION_BLOCK "Main"   // OB1, LAD, ProgramCycle
TITLE = "Main Program Sweep (Cycle)"
{ S7_Optimized_Access := 'TRUE' }
VERSION : 0.1
   VAR_TEMP
      Ret_Val : Int;
   END_VAR
BEGIN

REGION Network 1: Program główny szklarni
   // Główny algorytm działania programu.
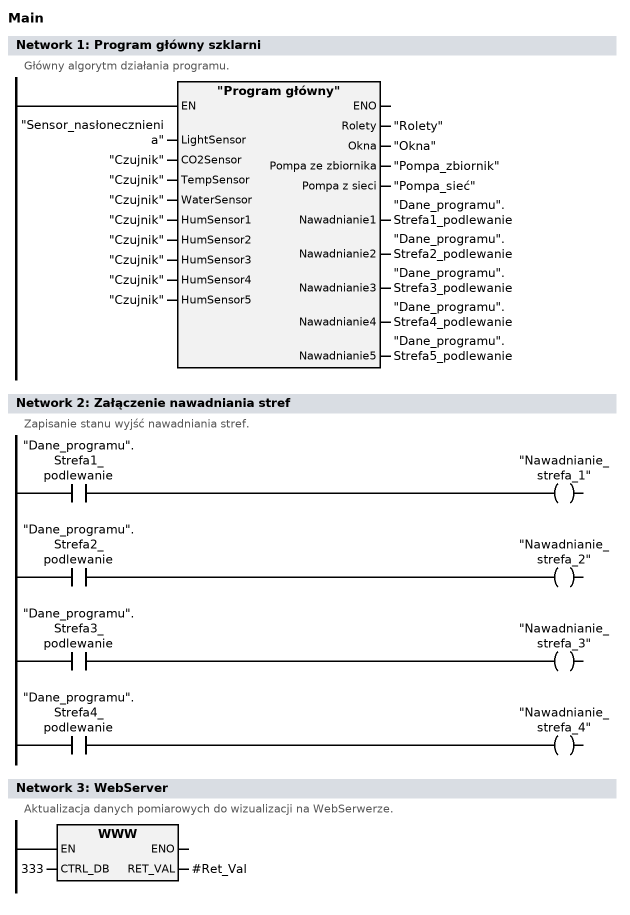
   RUNG wire#powerrail
      "Program główny"(LightSensor := "Sensor_nasłonecznienia", CO2Sensor := "Czujnik", TempSensor := "Czujnik", WaterSensor := "Czujnik", HumSensor1 := "Czujnik", HumSensor2 := "Czujnik", HumSensor3 := "Czujnik", HumSensor4 := "Czujnik", HumSensor5 := "Czujnik", Rolety => "Rolety", Okna => "Okna", "Pompa ze zbiornika" => "Pompa_zbiornik", "Pompa z sieci" => "Pompa_sieć", Nawadnianie1 => "Dane_programu".Strefa1_podlewanie, Nawadnianie2 => "Dane_programu".Strefa2_podlewanie, Nawadnianie3 => "Dane_programu".Strefa3_podlewanie, Nawadnianie4 => "Dane_programu".Strefa4_podlewanie, Nawadnianie5 => "Dane_programu".Strefa5_podlewanie)
   END_RUNG
   // the same network as SCL:
   "Program główny"(LightSensor := "Sensor_nasłonecznienia",
                    CO2Sensor := "Czujnik",
                    TempSensor := "Czujnik",
                    WaterSensor := "Czujnik",
                    HumSensor1 := "Czujnik",
                    HumSensor2 := "Czujnik",
                    HumSensor3 := "Czujnik",
                    HumSensor4 := "Czujnik",
                    HumSensor5 := "Czujnik",
                    Rolety => "Rolety",
                    Okna => "Okna",
                    "Pompa ze zbiornika" => "Pompa_zbiornik",
                    "Pompa z sieci" => "Pompa_sieć",
                    Nawadnianie1 => "Dane_programu".Strefa1_podlewanie,
                    Nawadnianie2 => "Dane_programu".Strefa2_podlewanie,
                    Nawadnianie3 => "Dane_programu".Strefa3_podlewanie,
                    Nawadnianie4 => "Dane_programu".Strefa4_podlewanie,
                    Nawadnianie5 => "Dane_programu".Strefa5_podlewanie);
END_REGION

REGION Network 2: Załączenie nawadniania stref
   // Zapisanie stanu wyjść nawadniania stref.
   RUNG wire#powerrail
      Contact( "Dane_programu".Strefa1_podlewanie )
      Coil( "Nawadnianie_strefa_1" )
   END_RUNG
   RUNG wire#powerrail
      Contact( "Dane_programu".Strefa2_podlewanie )
      Coil( "Nawadnianie_strefa_2" )
   END_RUNG
   RUNG wire#powerrail
      Contact( "Dane_programu".Strefa3_podlewanie )
      Coil( "Nawadnianie_strefa_3" )
   END_RUNG
   RUNG wire#powerrail
      Contact( "Dane_programu".Strefa4_podlewanie )
      Coil( "Nawadnianie_strefa_4" )
   END_RUNG
   // the same network as SCL:
   "Nawadnianie_strefa_1" := "Dane_programu".Strefa1_podlewanie;
   "Nawadnianie_strefa_2" := "Dane_programu".Strefa2_podlewanie;
   "Nawadnianie_strefa_3" := "Dane_programu".Strefa3_podlewanie;
   "Nawadnianie_strefa_4" := "Dane_programu".Strefa4_podlewanie;
END_REGION

REGION Network 3: WebServer
   // Aktualizacja danych pomiarowych do wizualizacji na WebSerwerze.
   #Ret_Val := WWW(CTRL_DB := 333);
END_REGION
END_ORGANIZATION_BLOCK

(* ===== HMI "HMI_RT_1" =====
system functions are stored by id; their names below are inferred from use
connection "HMI_Connection_1": ETHERNET, SMART_S7_1200_OMS

HMI tags "Default tag table"
   "Dane_programu_lightLux_" : Real = PLC Dane_programu.lightLux_, 1 s
   "Dane_programu_Temp_" : Real = PLC Dane_programu.Temp_, 1 s
   "Dane_programu_CO2_" : Real = PLC Dane_programu.CO2_, 1 s
   "Dane_programu_StopPodlewanie" : Bool = PLC Dane_programu.StopPodlewanie, 1 s
   "Dane_programu_blindShut" : Bool = PLC Dane_programu.blindShut, 1 s
   "Dane_programu_WinOpen" : Bool = PLC Dane_programu.WinOpen, 1 s
   "Dane_programu_StopBtn" : Bool = PLC Dane_programu.StopBtn, 1 s
   "Dane_programu_Strefa1" : Bool = PLC Dane_programu.Strefa1, 1 s
   "Dane_programu_Strefa2" : Bool = PLC Dane_programu.Strefa2, 1 s
   "Dane_programu_Strefa3" : Bool = PLC Dane_programu.Strefa3, 1 s
   "Dane_programu_Strefa4" : Bool = PLC Dane_programu.Strefa4, 1 s
   "Dane_programu_Strefa5" : Bool = PLC Dane_programu.Strefa5, 1 s
   "Dane_programu_Hum_Strefa1" : Real = PLC Dane_programu.Hum_Strefa1, 1 s
   "Dane_programu_Hum_Strefa2" : Real = PLC Dane_programu.Hum_Strefa2, 1 s
   "Dane_programu_Hum_Strefa3" : Real = PLC Dane_programu.Hum_Strefa3, 1 s
   "Dane_programu_Hum_Strefa4" : Real = PLC Dane_programu.Hum_Strefa4, 1 s
   "Dane_programu_Hum_Strefa5" : Real = PLC Dane_programu.Hum_Strefa5, 1 s
   "Dane_programu_setLux" : Real = PLC Dane_programu.setLux, 1 s
   "Dane_programu_setTemp" : Real = PLC Dane_programu.setTemp, 1 s
   "Dane_programu_setCO2" : Real = PLC Dane_programu.setCO2, 1 s
   "Dane_programu_setHum_Strefa1" : Real = PLC Dane_programu.setHum_Strefa1, 1 s
   "Dane_programu_setHum_Strefa2" : Real = PLC Dane_programu.setHum_Strefa2, 1 s
   "Dane_programu_setHum_Strefa3" : Real = PLC Dane_programu.setHum_Strefa3, 1 s
   "Dane_programu_Strefa1_podlewanie" : Bool = PLC Dane_programu.Strefa1_podlewanie, 1 s
   "Dane_programu_Strefa2_podlewanie" : Bool = PLC Dane_programu.Strefa2_podlewanie, 1 s
   "Dane_programu_Strefa3_podlewanie" : Bool = PLC Dane_programu.Strefa3_podlewanie, 1 s
   "Dane_programu_Strefa4_podlewanie" : Bool = PLC Dane_programu.Strefa4_podlewanie, 1 s
   "Dane_programu_Strefa5_podlewanie" : Bool = PLC Dane_programu.Strefa5_podlewanie, 1 s
   "Dane_programu_setLux_" : Real = PLC Dane_programu.setLux_, 1 s
   "Dane_programu_setTemp_" : Real = PLC Dane_programu.setTemp_, 1 s
   "Dane_programu_setCO2_" : Real = PLC Dane_programu.setCO2_, 1 s
   "Dane_programu_setHum_Strefa1_" : Real = PLC Dane_programu.setHum_Strefa1_, 1 s
   "Dane_programu_setHum_Strefa2_" : Real = PLC Dane_programu.setHum_Strefa2_, 1 s
   "Dane_programu_setHum_Strefa3_" : Real = PLC Dane_programu.setHum_Strefa3_, 1 s
   "Dane_programu_setHum_Strefa4_" : Real = PLC Dane_programu.setHum_Strefa4_, 1 s
   "Dane_programu_setHum_Strefa5_" : Real = PLC Dane_programu.setHum_Strefa5_, 1 s
   "Dane_programu_setCO2__" : Real = PLC Dane_programu.setCO2_, 1 s
   "Dane_programu_setHum_Strefa1__" : Real = PLC Dane_programu.setHum_Strefa1_, 1 s
   "Dane_programu_setHum_Strefa2__" : Real = PLC Dane_programu.setHum_Strefa2_, 1 s
   "Dane_programu_setHum_Strefa3__" : Real = PLC Dane_programu.setHum_Strefa3_, 1 s
   "Dane_programu_setHum_Strefa4__" : Real = PLC Dane_programu.setHum_Strefa4_, 1 s
   "Dane_programu_setHum_Strefa5__" : Real = PLC Dane_programu.setHum_Strefa5_, 1 s
   "Dane_programu_setLux__" : Real = PLC Dane_programu.setLux_, 1 s
   "Dane_programu_setTemp__" : Real = PLC Dane_programu.setTemp_, 1 s

recipe "Recipe_1": Temperatura <- "Dane_programu_setTemp__", CO2: <- "Dane_programu_setCO2__", Nasłonecznienie <- "Dane_programu_setLux__", Strefa 1 <- "Dane_programu_setHum_Strefa1__", Strefa 2 <- "Dane_programu_setHum_Strefa2__", Strefa 3 <- "Dane_programu_setHum_Strefa3__", Strefa 4 <- "Dane_programu_setHum_Strefa4__", Strefa 5 <- "Dane_programu_setHum_Strefa5__"

Template "Template_1" 320x240
   Button "Template_Button_2" at 0,201 size 74x37; TextOff 'ToggleLanguage'; PictureOff "ToggleLanguage_KTP600_Basic_color_PN"; PictureOn "ToggleLanguage_KTP600_Basic_color_PN"
      on Release: function_fb9197e8(-1)
   Button "Template_Button_5" at 0,163 size 73x37; TextOff 'Ustawienia / Einstellungen / Settings'; TextOn 'Ustawienia'
      on Press: ActivateScreen("Ustawienia", 0)
   Button "Template_Button_1" at 0,124 size 73x37; TextOff 'Nawadnianie / Bewasserung / Irrigation'; TextOn 'Ustawienia'
      on Press: ActivateScreen("Nawadnianie", 0)
   Button "Template_Button_3" at 0,85 size 73x37; TextOff 'Parametry / Parameter / Parameters'; TextOn 'Ustawienia'
      on Press: ActivateScreen("CO2,Temp", 0)
   Button "Template_Button_4" at 0,46 size 73x37; TextOff 'START'; TextOn 'Ustawienia'
      on Press: ActivateScreen("Home", 0)

screen "Home" 320x240, template "Template_1"
   TextField "Text field_1" at 0,0 size 319x47; Text 'Zautomatyzowana szklarnia / Automatisiertes Gewachshaus / Automated greenhouse'
   GraphicView "Graphic view_1" at 100,80 size 182x91; Picture "Logo_projekt"
   TextField "Text field_2" at 91,198 size 202x41; Text 'Agnieszka Piórkowska, Natalia Wiśniewska, Miłosz Gajewski'

screen "CO2,Temp" 320x240, template "Template_1"
   TextField "Text field_1" at 0,0 size 319x44; Text 'Nasłonecznienie, CO2, Temperatura / Sonneneinstrahlung, CO2, Temperatur / Insolation, CO2, Temperature'
   TextField "Text field_2" at 74,52 size 124x29; Text 'Nasłonecznienie: / Sosnneneinstrahlung / Insolation:'
   IOField "I/O field_1" at 202,57 size 45x23; FormatPattern 99
      ProcessValue <- "Dane_programu_lightLux_"
   TextField "Text field_3" at 277,57 size 20x20; Text '%'
   TextField "Text field_4" at 76,84 size 125x25; Text 'Temperatura: / Temperatur: / Temperature:'
   IOField "I/O field_2" at 202,88 size 46x23; FormatPattern 99
      ProcessValue <- "Dane_programu_Temp_"
   TextField "Text field_5" at 277,88 size 20x20; Text 'C / %'
   IOField "I/O field_3" at 201,119 size 47x23; FormatPattern 99
      ProcessValue <- "Dane_programu_CO2_"
   TextField "Text field_6" at 274,119 size 33x20; Text 'ppm / %'
   TextField "Text field_7" at 78,117 size 122x25; Text 'CO2:'
   Button "Button_1" at 76,155 size 115x28; TextOff 'Zablokuj podlewanie / Bewasserung blockieren / Lock watering'; TextOn 'Zablokuj podlewanie'
      on Press: SetBit("Dane_programu_StopPodlewanie")
   Button "Button_2" at 198,155 size 117x28; TextOff 'Odblokuj podlewanie / Bewasserung freischalten / Unlock watering'
      on Press: ResetBit("Dane_programu_StopPodlewanie")
   TextField "Text field_8" at 80,187 size 137x29; Text 'Rolety: / Rollos: / Blindes:'
   Circle "Circle_1" at 220,195 size 17x17
      Appearance <- "Dane_programu_blindShut"
   TextField "Text field_9" at 79,212 size 138x22; Text 'Okna: / Fenster: / Windows:'
   Circle "Circle_2" at 220,217 size 17x17
      Appearance <- "Dane_programu_WinOpen"
   Button "Button_3" at 258,190 size 56x44; TextOff 'STOP'
      on Press: InvertBit("Dane_programu_StopBtn")

screen "Nawadnianie" 320x240, template "Template_1"
   TextField "Text field_1" at 3,4 size 316x38; Text 'Nawadnianie / Bewasserung / Irrigation'
   TextField "Text field_2" at 83,65 size 46x13; Text 'Strefa 1: / Zone 1:'
   TextField "Text field_3" at 83,97 size 46x13; Text 'Strefa 2: / Zone 2:'
   TextField "Text field_4" at 84,128 size 46x13; Text 'Strefa 3: / Zone 3:'
   TextField "Text field_5" at 83,159 size 46x13; Text 'Strefa 4: / Zone 4:'
   TextField "Text field_6" at 83,190 size 46x13; Text 'Strefa 5: / Zone 5:'
   Circle "Circle_1" at 135,62 size 22x22
      Appearance <- "Dane_programu_Strefa1_podlewanie"
   Circle "Circle_2" at 135,93 size 22x22
      Appearance <- "Dane_programu_Strefa2_podlewanie"
   Circle "Circle_3" at 135,124 size 22x22
      Appearance <- "Dane_programu_Strefa3_podlewanie"
   Circle "Circle_4" at 135,155 size 22x22
      Appearance <- "Dane_programu_Strefa4_podlewanie"
   Circle "Circle_5" at 135,186 size 22x22
      Appearance <- "Dane_programu_Strefa5_podlewanie"
   TextField "Text field_7" at 167,63 size 75x15; Text 'Wiglotność: / Feuchtigkeit: / Humidity:'
   TextField "Text field_8" at 167,93 size 75x15; Text 'Wiglotność: / Feuchtigkeit: / Humidity:'
   TextField "Text field_9" at 167,93 size 75x15; Text 'Wiglotność: / Feuchtigkeit: / Humidity:'
   TextField "Text field_10" at 167,124 size 75x15; Text 'Wiglotność: / Feuchtigkeit: / Humidity:'
   TextField "Text field_11" at 167,155 size 75x15; Text 'Wiglotność: / Feuchtigkeit: / Humidity:'
   TextField "Text field_12" at 167,189 size 75x15; Text 'Wiglotność: / Feuchtigkeit: / Humidity:'
   IOField "I/O field_1" at 236,61 size 59x23; FormatPattern 99.9
      ProcessValue <- "Dane_programu_Hum_Strefa1"
   IOField "I/O field_2" at 236,93 size 59x23; FormatPattern 99.9
      ProcessValue <- "Dane_programu_Hum_Strefa2"
   IOField "I/O field_3" at 236,125 size 59x23; FormatPattern 99.9
      ProcessValue <- "Dane_programu_Hum_Strefa3"
   IOField "I/O field_4" at 236,157 size 59x23; FormatPattern 99.9
      ProcessValue <- "Dane_programu_Hum_Strefa4"
   IOField "I/O field_5" at 236,189 size 59x23; FormatPattern 99.9
      ProcessValue <- "Dane_programu_Hum_Strefa5"
   TextField "Text field_13" at 295,62 size 29x16; Text '%'
   TextField "Text field_14" at 296,94 size 29x16; Text '%'
   TextField "Text field_15" at 294,126 size 29x16; Text '%'
   TextField "Text field_16" at 294,158 size 29x16; Text '%'
   TextField "Text field_17" at 293,190 size 29x16; Text '%'
   Button "Button_1" at 76,210 size 27x26; TextOff '1'
      Appearance <- "Dane_programu_Strefa1"
      on Press: InvertBit("Dane_programu_Strefa1")
   Button "Button_2" at 103,210 size 29x26; TextOff '2'
      Appearance <- "Dane_programu_Strefa2"
      on Press: InvertBit("Dane_programu_Strefa2")
   Button "Button_3" at 132,210 size 27x26; TextOff '3'
      on Press: InvertBit("Dane_programu_Strefa3")
      Appearance <- "Dane_programu_Strefa3"
   Button "Button_4" at 159,210 size 27x26; TextOff '4'
      on Press: InvertBit("Dane_programu_Strefa4")
      Appearance <- "Dane_programu_Strefa4"
   Button "Button_5" at 186,210 size 27x26; TextOff '5'
      on Press: InvertBit("Dane_programu_Strefa5")
      Appearance <- "Dane_programu_Strefa5"

screen "Ustawienia" 320x240, template "Template_1"
   TextField "Text field_1" at 0,0 size 319x45; Text 'Ustawienia / Einstellungen / Settings'
   TextField "Text field_2" at 79,59 size 113x19; Text 'Nasłonecznienie: / Sosnneneinstrahlung / Insolation:'
   IOField "I/O field_1" at 202,57 size 45x23; FormatPattern 99
      ProcessValue <- "Dane_programu_setLux_"
   TextField "Text field_3" at 280,57 size 20x20; Text '%'
   TextField "Text field_4" at 80,91 size 115x16; Text 'Temperatura: / Temperatur: / Temperature:'
   IOField "I/O field_2" at 203,88 size 45x23; FormatPattern 99
      ProcessValue <- "Dane_programu_setTemp_"
   TextField "Text field_5" at 279,88 size 20x20; Text 'C / %'
   IOField "I/O field_3" at 203,119 size 45x23; FormatPattern 99
      ProcessValue <- "Dane_programu_setCO2_"
   TextField "Text field_7" at 78,117 size 117x26; Text 'CO2:'
   TextField "Text field_6" at 276,117 size 33x20; Text 'ppm'
   TextField "Text field_8" at 76,140 size 243x19; Text 'Nawadnianie / Bewasserung / Irrigation'
   TextField "Text field_9" at 87,168 size 46x13; Text 'Strefa 1: / Zone 1:'
   TextField "Text field_10" at 87,197 size 46x13; Text 'Strefa 2: / Zone 2:'
   TextField "Text field_11" at 88,221 size 46x13; Text 'Strefa 3: / Zone 3:'
   IOField "I/O field_4" at 137,165 size 48x22; FormatPattern 99
      ProcessValue <- "Dane_programu_setHum_Strefa1_"
   IOField "I/O field_5" at 137,190 size 48x22; FormatPattern 99
      ProcessValue <- "Dane_programu_setHum_Strefa2_"
   IOField "I/O field_6" at 137,214 size 48x22; FormatPattern 99
      ProcessValue <- "Dane_programu_setHum_Strefa3_"
   TextField "Text field_12" at 200,167 size 46x13; Text 'Strefa 4: / Zone 4:'
   TextField "Text field_13" at 200,196 size 46x13; Text 'Strefa 5: / Zone 5:'
   IOField "I/O field_7" at 250,164 size 48x22; FormatPattern 99
      ProcessValue <- "Dane_programu_setHum_Strefa4_"
   IOField "I/O field_8" at 250,189 size 48x22; FormatPattern 99
      ProcessValue <- "Dane_programu_setHum_Strefa5_"
   Button "Button_1" at 202,215 size 113x20; TextOff 'Przepisy / Recipes'
      on Click: ActivateScreen("Przepisy", 0)

screen "Przepisy" 320x240, template "Template_1"
   TextField "Text field_1" at 0,0 size 319x48; Text 'Przepisy / Recipes'
   RecipeView "Recipe view_1" at 76,50 size 240x188; Recipe "Recipe_1"
*)